Yaskawa INFORM job: DEMO_ROOF_UPPER_0625_3PAINT_69.JBI

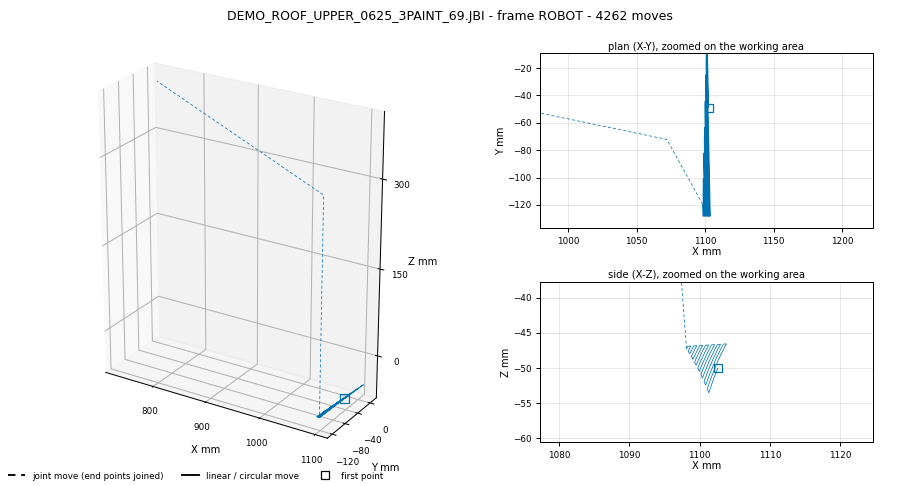
[picture p0: tool path of DEMO_ROOF_UPPER_0625_3PAINT_69.JBI in frame ROBOT, 4262 of 4262 moves have a stored position in this frame; points joined in program order, loops and branches not executed]
/JOB
//NAME DEMO_ROOF_UPPER_0625_3PAINT69
//POS
///NPOS 4262,0,0,0,0,0
///TOOL 0
///USER 0
///POSTYPE ROBOT
///RECTAN
///RCONF 1,0,0,0,0,0,0,0,0,0,0,0,0,0,0,0,0,0,0,0,0,0,0,0
C00000=1102.592,-48.864,-50.002,179.869,5.615,149.029
C00001=1102.586,-48.614,-50.014,179.869,5.619,149.030
C00002=1102.581,-48.364,-50.026,179.869,5.624,149.031
C00003=1102.575,-48.115,-50.039,179.869,5.629,149.032
C00004=1102.571,-47.865,-50.052,179.869,5.633,149.033
C00005=1102.566,-47.615,-50.065,179.868,5.638,149.034
C00006=1102.560,-47.366,-50.078,179.868,5.643,149.035
C00007=1102.555,-47.116,-50.090,179.868,5.648,149.037
C00008=1102.550,-46.866,-50.103,179.868,5.652,149.037
C00009=1102.545,-46.617,-50.115,179.868,5.657,149.039
C00010=1102.540,-46.368,-50.128,179.867,5.661,149.040
C00011=1102.534,-46.118,-50.141,179.868,5.666,149.041
C00012=1102.530,-45.904,-50.152,179.867,5.670,149.042
C00013=1102.526,-45.689,-50.162,179.867,5.674,149.043
C00014=1102.522,-45.475,-50.174,179.867,5.678,149.044
C00015=1102.517,-45.261,-50.184,179.867,5.683,149.045
C00016=1102.513,-45.047,-50.195,179.867,5.687,149.046
C00017=1102.508,-44.833,-50.206,179.867,5.691,149.046
C00018=1102.504,-44.618,-50.217,179.867,5.695,149.047
C00019=1102.500,-44.405,-50.228,179.866,5.699,149.048
C00020=1102.494,-44.154,-50.241,179.866,5.704,149.049
C00021=1102.489,-43.905,-50.253,179.866,5.708,149.050
C00022=1102.484,-43.656,-50.266,179.866,5.713,149.051
C00023=1102.479,-43.406,-50.279,179.866,5.718,149.053
C00024=1102.474,-43.157,-50.291,179.865,5.722,149.054
C00025=1102.468,-42.907,-50.305,179.866,5.727,149.055
C00026=1102.464,-42.657,-50.318,179.865,5.731,149.056
C00027=1102.459,-42.408,-50.330,179.865,5.737,149.057
C00028=1102.454,-42.158,-50.343,179.866,5.741,149.058
C00029=1102.449,-41.908,-50.356,179.866,5.746,149.059
C00030=1102.443,-41.659,-50.369,179.865,5.750,149.060
C00031=1102.438,-41.409,-50.382,179.865,5.756,149.061
C00032=1102.433,-41.160,-50.394,179.866,5.760,149.062
C00033=1102.428,-40.910,-50.407,179.866,5.765,149.063
C00034=1102.423,-40.660,-50.420,179.866,5.769,149.064
C00035=1102.417,-40.411,-50.433,179.865,5.774,149.065
C00036=1102.413,-40.161,-50.446,179.866,5.779,149.066
C00037=1102.407,-39.911,-50.459,179.866,5.783,149.067
C00038=1102.402,-39.662,-50.472,179.866,5.788,149.068
C00039=1102.397,-39.412,-50.485,179.866,5.793,149.069
C00040=1102.393,-39.163,-50.498,179.866,5.797,149.070
C00041=1102.387,-38.913,-50.512,179.866,5.802,149.071
C00042=1102.382,-38.664,-50.524,179.867,5.806,149.072
C00043=1102.377,-38.414,-50.537,179.867,5.811,149.073
C00044=1102.372,-38.164,-50.550,179.867,5.815,149.074
C00045=1102.367,-37.915,-50.563,179.867,5.820,149.075
C00046=1102.362,-37.665,-50.576,179.868,5.825,149.076
C00047=1102.356,-37.415,-50.589,179.867,5.829,149.077
C00048=1102.351,-37.166,-50.602,179.868,5.834,149.078
C00049=1102.346,-36.916,-50.616,179.868,5.837,149.079
C00050=1102.341,-36.667,-50.629,179.868,5.842,149.079
C00051=1102.336,-36.417,-50.641,179.869,5.847,149.080
C00052=1102.331,-36.167,-50.655,179.868,5.851,149.081
C00053=1102.326,-35.918,-50.667,179.869,5.856,149.082
C00054=1102.321,-35.668,-50.681,179.869,5.860,149.083
C00055=1102.316,-35.419,-50.694,179.869,5.864,149.084
C00056=1102.310,-35.169,-50.707,179.870,5.869,149.085
C00057=1102.305,-34.919,-50.720,179.870,5.874,149.086
C00058=1102.300,-34.670,-50.733,179.870,5.878,149.087
C00059=1102.296,-34.420,-50.747,179.870,5.882,149.088
C00060=1102.290,-34.171,-50.760,179.871,5.887,149.089
C00061=1102.285,-33.921,-50.773,179.871,5.891,149.089
C00062=1102.280,-33.671,-50.786,179.871,5.896,149.090
C00063=1102.275,-33.422,-50.799,179.872,5.901,149.091
C00064=1102.270,-33.172,-50.813,179.871,5.904,149.092
C00065=1102.264,-32.923,-50.825,179.872,5.909,149.093
C00066=1102.260,-32.673,-50.839,179.873,5.914,149.094
C00067=1102.254,-32.424,-50.852,179.873,5.917,149.095
C00068=1102.250,-32.209,-50.863,179.873,5.922,149.096
C00069=1102.246,-31.996,-50.875,179.874,5.926,149.096
C00070=1102.241,-31.781,-50.886,179.874,5.929,149.097
C00071=1102.237,-31.567,-50.898,179.874,5.933,149.098
C00072=1102.233,-31.353,-50.909,179.874,5.937,149.099
C00073=1102.229,-31.139,-50.921,179.875,5.941,149.099
C00074=1102.224,-30.925,-50.932,179.875,5.945,149.100
C00075=1102.220,-30.711,-50.944,179.875,5.949,149.101
C00076=1102.214,-30.461,-50.957,179.876,5.953,149.102
C00077=1102.210,-30.212,-50.971,179.876,5.957,149.103
C00078=1102.204,-29.962,-50.983,179.876,5.962,149.104
C00079=1102.199,-29.712,-50.997,179.876,5.967,149.104
C00080=1102.194,-29.463,-51.010,179.877,5.971,149.105
C00081=1102.189,-29.213,-51.024,179.877,5.975,149.106
C00082=1102.184,-28.964,-51.037,179.877,5.980,149.107
C00083=1102.179,-28.714,-51.051,179.878,5.984,149.108
C00084=1102.174,-28.465,-51.064,179.879,5.989,149.109
C00085=1102.169,-28.215,-51.078,179.879,5.994,149.110
C00086=1102.164,-27.966,-51.091,179.879,5.998,149.111
C00087=1102.159,-27.716,-51.105,179.879,6.003,149.112
C00088=1102.153,-27.467,-51.118,179.879,6.008,149.113
C00089=1102.149,-27.217,-51.131,179.880,6.012,149.114
C00090=1102.143,-26.967,-51.145,179.880,6.017,149.114
C00091=1102.139,-26.718,-51.158,179.881,6.022,149.115
C00092=1102.134,-26.468,-51.173,179.881,6.027,149.116
C00093=1102.128,-26.219,-51.186,179.881,6.030,149.117
C00094=1102.124,-25.969,-51.199,179.882,6.035,149.118
C00095=1102.118,-25.720,-51.213,179.882,6.040,149.119
C00096=1102.114,-25.470,-51.226,179.883,6.045,149.120
C00097=1102.108,-25.220,-51.240,179.883,6.050,149.121
C00098=1102.103,-24.971,-51.254,179.883,6.054,149.122
C00099=1102.098,-24.721,-51.267,179.883,6.058,149.123
C00100=1102.093,-24.472,-51.281,179.883,6.064,149.124
C00101=1102.088,-24.222,-51.295,179.883,6.068,149.125
C00102=1102.083,-23.972,-51.308,179.884,6.073,149.126
C00103=1102.078,-23.723,-51.322,179.884,6.078,149.127
C00104=1102.072,-23.473,-51.335,179.884,6.082,149.128
C00105=1102.068,-23.224,-51.349,179.884,6.087,149.129
C00106=1102.063,-22.974,-51.363,179.885,6.091,149.130
C00107=1102.057,-22.724,-51.377,179.885,6.096,149.131
C00108=1102.052,-22.475,-51.390,179.885,6.100,149.131
C00109=1102.048,-22.226,-51.404,179.886,6.105,149.132
C00110=1102.042,-21.975,-51.418,179.886,6.110,149.133
C00111=1102.037,-21.726,-51.432,179.886,6.115,149.134
C00112=1102.033,-21.477,-51.445,179.886,6.119,149.135
C00113=1102.027,-21.227,-51.458,179.886,6.123,149.136
C00114=1102.022,-20.977,-51.473,179.887,6.128,149.137
C00115=1102.017,-20.728,-51.487,179.887,6.133,149.138
C00116=1102.012,-20.478,-51.500,179.887,6.137,149.139
C00117=1102.007,-20.229,-51.514,179.888,6.141,149.140
C00118=1102.002,-19.979,-51.528,179.888,6.147,149.141
C00119=1101.996,-19.730,-51.542,179.888,6.151,149.142
C00120=1101.991,-19.480,-51.556,179.889,6.156,149.143
C00121=1101.987,-19.230,-51.569,179.889,6.160,149.144
C00122=1101.981,-18.981,-51.583,179.889,6.165,149.145
C00123=1101.976,-18.732,-51.598,179.890,6.169,149.145
C00124=1101.972,-18.518,-51.610,179.890,6.173,149.146
C00125=1101.967,-18.304,-51.622,179.890,6.177,149.147
C00126=1101.963,-18.090,-51.634,179.891,6.181,149.148
C00127=1101.959,-17.876,-51.645,179.891,6.185,149.149
C00128=1101.954,-17.662,-51.656,179.891,6.189,149.149
C00129=1101.950,-17.447,-51.669,179.891,6.192,149.150
C00130=1101.946,-17.233,-51.681,179.891,6.196,149.151
C00131=1101.942,-17.019,-51.693,179.892,6.200,149.152
C00132=1101.936,-16.770,-51.707,179.892,6.204,149.152
C00133=1101.931,-16.520,-51.721,179.893,6.209,149.153
C00134=1101.927,-16.271,-51.735,179.893,6.214,149.154
C00135=1101.922,-16.021,-51.749,179.894,6.218,149.155
C00136=1101.916,-15.772,-51.763,179.894,6.223,149.156
C00137=1101.911,-15.523,-51.777,179.894,6.227,149.157
C00138=1101.906,-15.273,-51.791,179.894,6.232,149.158
C00139=1101.901,-15.023,-51.805,179.895,6.237,149.159
C00140=1101.896,-14.774,-51.819,179.895,6.241,149.160
C00141=1101.891,-14.524,-51.833,179.896,6.246,149.161
C00142=1101.886,-14.274,-51.847,179.896,6.250,149.161
C00143=1101.881,-14.025,-51.861,179.897,6.254,149.162
C00144=1101.876,-13.776,-51.875,179.897,6.259,149.163
C00145=1101.871,-13.526,-51.889,179.898,6.264,149.164
C00146=1101.866,-13.276,-51.904,179.898,6.268,149.165
C00147=1101.861,-13.027,-51.918,179.898,6.272,149.166
C00148=1101.856,-12.777,-51.932,179.899,6.277,149.167
C00149=1101.850,-12.528,-51.946,179.899,6.282,149.168
C00150=1101.846,-12.278,-51.960,179.900,6.286,149.168
C00151=1101.841,-12.028,-51.975,179.900,6.290,149.169
C00152=1101.836,-11.779,-51.989,179.901,6.295,149.170
C00153=1101.831,-11.529,-52.003,179.901,6.299,149.171
C00154=1101.825,-11.280,-52.017,179.902,6.304,149.172
C00155=1101.820,-11.030,-52.031,179.902,6.309,149.173
C00156=1101.815,-10.781,-52.046,179.903,6.314,149.174
C00157=1101.811,-10.531,-52.061,179.903,6.317,149.174
C00158=1101.806,-10.282,-52.075,179.903,6.322,149.175
C00159=1101.801,-10.032,-52.089,179.904,6.327,149.176
C00160=1101.795,-9.783,-52.103,179.905,6.331,149.177
C00161=1101.790,-9.533,-52.117,179.905,6.336,149.178
C00162=1101.785,-9.284,-52.132,179.905,6.340,149.179
C00163=1101.780,-9.034,-52.146,179.906,6.344,149.179
C00164=1101.775,-8.784,-52.160,179.906,6.349,149.180
C00165=1101.770,-8.535,-52.175,179.907,6.354,149.181
C00166=1101.766,-8.285,-52.189,179.907,6.358,149.182
C00167=1101.760,-8.036,-52.203,179.908,6.363,149.183
C00168=1101.755,-7.787,-52.218,179.908,6.367,149.184
C00169=1101.750,-7.537,-52.232,179.909,6.371,149.185
C00170=1101.745,-7.287,-52.246,179.909,6.376,149.186
C00171=1101.741,-7.038,-52.261,179.910,6.380,149.186
C00172=1101.736,-6.788,-52.276,179.911,6.385,149.187
C00173=1101.730,-6.538,-52.290,179.911,6.390,149.188
C00174=1101.725,-6.289,-52.305,179.912,6.395,149.189
C00175=1101.720,-6.039,-52.319,179.912,6.398,149.190
C00176=1101.715,-5.791,-52.334,179.913,6.403,149.190
C00177=1101.710,-5.541,-52.348,179.913,6.408,149.191
C00178=1101.705,-5.291,-52.362,179.914,6.412,149.192
C00179=1101.700,-5.042,-52.377,179.915,6.417,149.193
C00180=1101.696,-4.828,-52.389,179.915,6.420,149.194
C00181=1101.691,-4.613,-52.402,179.916,6.425,149.194
C00182=1101.687,-4.400,-52.415,179.916,6.428,149.195
C00183=1101.683,-4.186,-52.427,179.916,6.432,149.196
C00184=1101.678,-3.973,-52.440,179.917,6.436,149.196
C00185=1101.675,-3.758,-52.452,179.918,6.440,149.197
C00186=1101.670,-3.544,-52.464,179.918,6.444,149.198
C00187=1101.666,-3.331,-52.477,179.919,6.448,149.199
C00188=1101.660,-3.081,-52.492,179.919,6.452,149.199
C00189=1101.656,-2.832,-52.507,179.920,6.456,149.200
C00190=1101.651,-2.582,-52.521,179.920,6.461,149.201
C00191=1101.646,-2.332,-52.535,179.921,6.466,149.202
C00192=1101.640,-2.083,-52.551,179.922,6.470,149.203
C00193=1101.635,-1.833,-52.565,179.922,6.475,149.204
C00194=1101.631,-1.584,-52.580,179.923,6.479,149.205
C00195=1101.626,-1.334,-52.594,179.924,6.484,149.205
C00196=1101.620,-1.084,-52.609,179.924,6.488,149.206
C00197=1101.615,-0.835,-52.624,179.925,6.493,149.207
C00198=1101.610,-0.586,-52.639,179.925,6.498,149.208
C00199=1101.606,-0.337,-52.654,179.926,6.502,149.209
C00200=1101.600,-0.086,-52.668,179.927,6.507,149.209
C00201=1101.595,0.163,-52.683,179.927,6.511,149.210
C00202=1101.590,0.412,-52.698,179.928,6.515,149.211
C00203=1101.586,0.661,-52.713,179.928,6.520,149.212
C00204=1101.580,0.911,-52.728,179.929,6.525,149.213
C00205=1101.575,1.161,-52.743,179.930,6.529,149.213
C00206=1101.571,1.410,-52.757,179.930,6.534,149.214
C00207=1101.565,1.660,-52.772,179.931,6.538,149.215
C00208=1101.560,1.909,-52.787,179.931,6.543,149.216
C00209=1101.556,2.158,-52.802,179.932,6.547,149.217
C00210=1101.550,2.408,-52.817,179.933,6.552,149.218
C00211=1101.545,2.658,-52.832,179.934,6.557,149.219
C00212=1101.541,2.907,-52.847,179.935,6.561,149.219
C00213=1101.535,3.157,-52.861,179.935,6.566,149.220
C00214=1101.530,3.406,-52.876,179.936,6.570,149.221
C00215=1101.526,3.656,-52.891,179.936,6.575,149.222
C00216=1101.520,3.906,-52.907,179.937,6.580,149.223
C00217=1101.516,4.155,-52.922,179.938,6.584,149.224
C00218=1101.510,4.405,-52.936,179.938,6.589,149.224
C00219=1101.505,4.654,-52.951,179.939,6.593,149.225
C00220=1101.501,4.903,-52.966,179.940,6.598,149.226
C00221=1101.495,5.153,-52.981,179.940,6.603,149.227
C00222=1101.490,5.402,-52.996,179.941,6.607,149.228
C00223=1101.485,5.651,-53.012,179.942,6.612,149.228
C00224=1101.480,5.901,-53.026,179.942,6.616,149.229
C00225=1101.475,6.151,-53.042,179.943,6.621,149.230
C00226=1101.471,6.400,-53.057,179.944,6.625,149.231
C00227=1101.466,6.649,-53.072,179.944,6.630,149.232
C00228=1101.460,6.899,-53.087,179.946,6.636,149.233
C00229=1101.456,7.148,-53.102,179.946,6.640,149.234
C00230=1101.450,7.398,-53.118,179.947,6.645,149.234
C00231=1101.446,7.647,-53.133,179.948,6.649,149.235
C00232=1101.441,7.898,-53.148,179.948,6.654,149.236
C00233=1101.436,8.147,-53.163,179.949,6.659,149.237
C00234=1101.431,8.396,-53.178,179.950,6.663,149.238
C00235=1101.426,8.645,-53.193,179.950,6.668,149.238
C00236=1101.419,8.979,-53.214,179.951,6.674,149.240
C00237=1101.412,9.313,-53.234,179.951,6.680,149.241
C00238=1101.406,9.648,-53.255,179.952,6.686,149.242
C00239=1101.399,9.982,-53.276,179.952,6.692,149.243
C00240=1101.394,10.231,-53.291,179.952,6.696,149.244
C00241=1101.388,10.481,-53.306,179.953,6.701,149.245
C00242=1101.384,10.730,-53.321,179.953,6.705,149.246
C00243=1101.379,10.980,-53.337,179.953,6.709,149.247
C00244=1101.374,11.229,-53.351,179.954,6.714,149.248
C00245=1101.369,11.478,-53.367,179.954,6.718,149.249
C00246=1101.364,11.728,-53.383,179.954,6.723,149.250
C00247=1101.359,11.978,-53.398,179.954,6.727,149.250
C00248=1101.354,12.227,-53.414,179.955,6.731,149.251
C00249=1101.349,12.476,-53.429,179.955,6.736,149.252
C00250=1101.344,12.725,-53.444,179.956,6.739,149.253
C00251=1101.339,12.975,-53.460,179.956,6.744,149.254
C00252=1101.335,13.225,-53.475,179.957,6.749,149.255
C00253=1101.329,13.474,-53.491,179.957,6.753,149.256
C00254=1101.325,13.723,-53.506,179.957,6.757,149.256
C00255=1101.319,13.973,-53.521,179.957,6.761,149.257
C00256=1101.094,4.203,-52.967,179.943,6.589,149.223
C00257=1101.098,3.953,-52.951,179.943,6.584,149.222
C00258=1101.102,3.704,-52.936,179.942,6.579,149.221
C00259=1101.108,3.454,-52.921,179.941,6.575,149.220
C00260=1101.113,3.205,-52.906,179.941,6.570,149.219
C00261=1101.118,2.956,-52.891,179.940,6.565,149.219
C00262=1101.123,2.706,-52.876,179.940,6.561,149.218
C00263=1101.128,2.457,-52.861,179.939,6.556,149.217
C00264=1101.133,2.207,-52.847,179.938,6.552,149.216
C00265=1101.138,1.958,-52.832,179.938,6.547,149.215
C00266=1101.143,1.709,-52.817,179.937,6.543,149.215
C00267=1101.148,1.459,-52.802,179.936,6.538,149.214
C00268=1101.153,1.209,-52.787,179.936,6.533,149.213
C00269=1101.158,0.960,-52.772,179.935,6.529,149.212
C00270=1101.163,0.710,-52.757,179.934,6.524,149.211
C00271=1101.168,0.461,-52.743,179.933,6.520,149.210
C00272=1101.173,0.212,-52.728,179.933,6.515,149.209
C00273=1101.178,-0.039,-52.712,179.932,6.511,149.209
C00274=1101.183,-0.288,-52.697,179.931,6.506,149.208
C00275=1101.188,-0.538,-52.683,179.931,6.501,149.207
C00276=1101.192,-0.787,-52.668,179.930,6.497,149.206
C00277=1101.198,-1.037,-52.653,179.929,6.492,149.205
C00278=1101.203,-1.286,-52.638,179.929,6.487,149.205
C00279=1101.208,-1.536,-52.624,179.928,6.483,149.204
C00280=1101.212,-1.785,-52.609,179.927,6.478,149.203
C00281=1101.218,-2.035,-52.594,179.927,6.474,149.202
C00282=1101.223,-2.285,-52.580,179.927,6.470,149.201
C00283=1101.228,-2.534,-52.565,179.926,6.465,149.201
C00284=1101.233,-2.783,-52.551,179.925,6.461,149.200
C00285=1101.239,-3.032,-52.535,179.925,6.456,149.199
C00286=1101.244,-3.282,-52.521,179.924,6.452,149.198
C00287=1101.248,-3.532,-52.507,179.923,6.447,149.197
C00288=1101.253,-3.781,-52.492,179.923,6.442,149.196
C00289=1101.260,-4.095,-52.474,179.922,6.436,149.195
C00290=1101.266,-4.408,-52.455,179.921,6.431,149.194
C00291=1101.273,-4.721,-52.437,179.921,6.426,149.193
C00292=1101.278,-5.034,-52.419,179.920,6.420,149.192
C00293=1101.283,-5.284,-52.404,179.919,6.415,149.191
C00294=1101.288,-5.533,-52.389,179.919,6.411,149.190
C00295=1101.294,-5.783,-52.374,179.918,6.406,149.190
C00296=1101.299,-6.033,-52.360,179.918,6.401,149.189
C00297=1101.304,-6.283,-52.346,179.917,6.397,149.188
C00298=1101.308,-6.532,-52.331,179.916,6.392,149.187
C00299=1101.314,-6.781,-52.317,179.916,6.388,149.186
C00300=1101.319,-7.030,-52.303,179.916,6.384,149.185
C00301=1101.324,-7.280,-52.288,179.915,6.379,149.185
C00302=1101.328,-7.529,-52.273,179.914,6.375,149.184
C00303=1101.333,-7.779,-52.259,179.914,6.370,149.183
C00304=1101.339,-8.029,-52.244,179.913,6.365,149.182
C00305=1101.344,-8.279,-52.230,179.913,6.362,149.181
C00306=1101.349,-8.528,-52.216,179.912,6.357,149.180
C00307=1101.354,-8.777,-52.201,179.912,6.352,149.179
C00308=1101.359,-9.026,-52.187,179.911,6.348,149.179
C00309=1101.364,-9.276,-52.173,179.911,6.343,149.178
C00310=1101.369,-9.526,-52.158,179.910,6.338,149.177
C00311=1101.374,-9.776,-52.144,179.910,6.335,149.176
C00312=1101.379,-10.025,-52.130,179.910,6.330,149.175
C00313=1101.384,-10.275,-52.115,179.909,6.325,149.174
C00314=1101.389,-10.524,-52.100,179.909,6.320,149.173
C00315=1101.394,-10.773,-52.087,179.908,6.316,149.173
C00316=1101.399,-11.023,-52.072,179.908,6.312,149.172
C00317=1101.404,-11.273,-52.058,179.907,6.307,149.171
C00318=1101.409,-11.522,-52.044,179.907,6.303,149.170
C00319=1101.414,-11.772,-52.029,179.906,6.298,149.169
C00320=1101.419,-12.022,-52.015,179.906,6.293,149.168
C00321=1101.424,-12.271,-52.001,179.905,6.290,149.168
C00322=1101.429,-12.520,-51.987,179.905,6.285,149.167
C00323=1101.434,-12.770,-51.973,179.904,6.280,149.166
C00324=1101.439,-13.020,-51.958,179.904,6.276,149.165
C00325=1101.444,-13.270,-51.944,179.903,6.271,149.164
C00326=1101.450,-13.519,-51.930,179.903,6.267,149.163
C00327=1101.455,-13.768,-51.916,179.903,6.262,149.162
C00328=1101.460,-14.018,-51.902,179.902,6.258,149.161
C00329=1101.464,-14.267,-51.888,179.901,6.253,149.161
C00330=1101.469,-14.517,-51.874,179.901,6.248,149.160
C00331=1101.474,-14.766,-51.860,179.901,6.245,149.159
C00332=1101.479,-15.016,-51.846,179.901,6.240,149.158
C00333=1101.484,-15.265,-51.831,179.900,6.235,149.157
C00334=1101.489,-15.515,-51.817,179.900,6.230,149.156
C00335=1101.495,-15.764,-51.803,179.899,6.226,149.155
C00336=1101.500,-16.014,-51.789,179.899,6.222,149.154
C00337=1101.505,-16.264,-51.775,179.899,6.217,149.153
C00338=1101.509,-16.514,-51.762,179.898,6.212,149.152
C00339=1101.515,-16.763,-51.748,179.898,6.208,149.152
C00340=1101.520,-17.012,-51.733,179.898,6.204,149.151
C00341=1101.524,-17.226,-51.721,179.897,6.199,149.150
C00342=1101.529,-17.440,-51.709,179.897,6.195,149.149
C00343=1101.533,-17.654,-51.697,179.897,6.192,149.148
C00344=1101.538,-17.868,-51.685,179.896,6.188,149.148
C00345=1101.542,-18.082,-51.673,179.896,6.184,149.147
C00346=1101.546,-18.296,-51.662,179.895,6.180,149.146
C00347=1101.550,-18.510,-51.649,179.895,6.176,149.145
C00348=1101.554,-18.724,-51.637,179.895,6.173,149.145
C00349=1101.560,-18.973,-51.623,179.895,6.168,149.144
C00350=1101.565,-19.223,-51.609,179.894,6.163,149.143
C00351=1101.570,-19.473,-51.596,179.894,6.159,149.142
C00352=1101.575,-19.722,-51.582,179.894,6.154,149.141
C00353=1101.580,-19.972,-51.568,179.894,6.149,149.140
C00354=1101.585,-20.221,-51.554,179.893,6.145,149.139
C00355=1101.590,-20.470,-51.540,179.893,6.140,149.138
C00356=1101.595,-20.721,-51.526,179.893,6.136,149.137
C00357=1101.600,-20.970,-51.513,179.892,6.131,149.136
C00358=1101.605,-21.219,-51.499,179.892,6.127,149.135
C00359=1101.610,-21.469,-51.485,179.891,6.122,149.134
C00360=1101.615,-21.719,-51.471,179.892,6.118,149.133
C00361=1101.620,-21.968,-51.458,179.892,6.113,149.132
C00362=1101.625,-22.218,-51.443,179.891,6.108,149.131
C00363=1101.630,-22.468,-51.430,179.891,6.103,149.131
C00364=1101.635,-22.717,-51.416,179.891,6.099,149.130
C00365=1101.640,-22.966,-51.402,179.890,6.095,149.129
C00366=1101.646,-23.216,-51.389,179.890,6.090,149.128
C00367=1101.651,-23.466,-51.375,179.890,6.085,149.127
C00368=1101.655,-23.715,-51.361,179.890,6.081,149.126
C00369=1101.661,-23.965,-51.348,179.889,6.076,149.125
C00370=1101.666,-24.214,-51.333,179.889,6.072,149.124
C00371=1101.671,-24.464,-51.320,179.889,6.066,149.123
C00372=1101.676,-24.713,-51.307,179.889,6.062,149.122
C00373=1101.681,-24.963,-51.292,179.889,6.058,149.121
C00374=1101.686,-25.212,-51.280,179.888,6.053,149.120
C00375=1101.691,-25.462,-51.265,179.888,6.048,149.119
C00376=1101.696,-25.712,-51.252,179.888,6.044,149.118
C00377=1101.701,-25.961,-51.239,179.888,6.039,149.117
C00378=1101.707,-26.211,-51.225,179.887,6.035,149.116
C00379=1101.712,-26.460,-51.211,179.887,6.030,149.115
C00380=1101.716,-26.710,-51.197,179.886,6.025,149.114
C00381=1101.722,-26.960,-51.184,179.886,6.020,149.113
C00382=1101.726,-27.209,-51.170,179.886,6.015,149.112
C00383=1101.732,-27.459,-51.157,179.885,6.011,149.111
C00384=1101.737,-27.708,-51.143,179.885,6.006,149.111
C00385=1101.742,-27.958,-51.130,179.885,6.001,149.110
C00386=1101.747,-28.207,-51.116,179.885,5.997,149.109
C00387=1101.752,-28.457,-51.103,179.884,5.992,149.108
C00388=1101.757,-28.706,-51.089,179.884,5.988,149.107
C00389=1101.762,-28.956,-51.076,179.883,5.983,149.106
C00390=1101.768,-29.206,-51.063,179.882,5.979,149.105
C00391=1101.773,-29.456,-51.049,179.882,5.975,149.104
C00392=1101.778,-29.705,-51.036,179.882,5.970,149.104
C00393=1101.783,-29.955,-51.022,179.882,5.965,149.103
C00394=1101.787,-30.205,-51.009,179.881,5.960,149.102
C00395=1101.793,-30.454,-50.995,179.881,5.956,149.101
C00396=1101.797,-30.704,-50.982,179.881,5.952,149.100
C00397=1101.802,-30.917,-50.970,179.880,5.948,149.099
C00398=1101.806,-31.131,-50.960,179.880,5.944,149.098
C00399=1101.811,-31.345,-50.948,179.880,5.940,149.098
C00400=1101.816,-31.560,-50.936,179.879,5.936,149.097
C00401=1101.819,-31.773,-50.925,179.879,5.933,149.096
C00402=1101.824,-31.988,-50.914,179.879,5.929,149.095
C00403=1101.828,-32.201,-50.902,179.878,5.925,149.095
C00404=1101.833,-32.416,-50.891,179.878,5.921,149.094
C00405=1101.838,-32.665,-50.878,179.878,5.917,149.093
C00406=1101.843,-32.915,-50.864,179.878,5.912,149.092
C00407=1101.848,-33.164,-50.851,179.877,5.908,149.091
C00408=1101.853,-33.414,-50.837,179.877,5.904,149.090
C00409=1101.858,-33.663,-50.825,179.877,5.899,149.089
C00410=1101.863,-33.914,-50.811,179.876,5.894,149.089
C00411=1101.868,-34.163,-50.798,179.876,5.890,149.088
C00412=1101.873,-34.413,-50.784,179.876,5.886,149.087
C00413=1101.878,-34.662,-50.771,179.875,5.881,149.086
C00414=1101.884,-34.911,-50.759,179.876,5.877,149.085
C00415=1101.889,-35.162,-50.745,179.875,5.872,149.084
C00416=1101.894,-35.410,-50.732,179.875,5.868,149.083
C00417=1101.899,-35.661,-50.718,179.875,5.864,149.082
C00418=1101.904,-35.910,-50.706,179.874,5.859,149.081
C00419=1101.909,-36.160,-50.693,179.874,5.854,149.080
C00420=1101.914,-36.409,-50.679,179.874,5.850,149.079
C00421=1101.919,-36.658,-50.666,179.874,5.845,149.078
C00422=1101.924,-36.909,-50.653,179.873,5.841,149.078
C00423=1101.930,-37.158,-50.640,179.873,5.837,149.077
C00424=1101.934,-37.408,-50.627,179.873,5.832,149.076
C00425=1101.940,-37.658,-50.614,179.873,5.828,149.075
C00426=1101.945,-37.906,-50.601,179.873,5.823,149.074
C00427=1101.949,-38.156,-50.588,179.872,5.819,149.073
C00428=1101.955,-38.406,-50.575,179.873,5.814,149.072
C00429=1101.960,-38.656,-50.562,179.872,5.810,149.071
C00430=1101.965,-38.905,-50.549,179.872,5.805,149.070
C00431=1101.971,-39.155,-50.536,179.872,5.801,149.069
C00432=1101.975,-39.405,-50.523,179.872,5.796,149.068
C00433=1101.980,-39.654,-50.510,179.872,5.791,149.067
C00434=1101.986,-39.903,-50.496,179.872,5.787,149.066
C00435=1101.990,-40.153,-50.483,179.871,5.782,149.065
C00436=1101.996,-40.403,-50.471,179.871,5.777,149.064
C00437=1102.001,-40.652,-50.458,179.872,5.773,149.063
C00438=1102.006,-40.902,-50.445,179.872,5.768,149.062
C00439=1102.011,-41.152,-50.432,179.871,5.764,149.061
C00440=1102.016,-41.401,-50.419,179.872,5.759,149.060
C00441=1102.021,-41.651,-50.406,179.871,5.754,149.059
C00442=1102.027,-41.901,-50.393,179.872,5.749,149.058
C00443=1102.032,-42.150,-50.381,179.871,5.745,149.057
C00444=1102.036,-42.400,-50.368,179.872,5.740,149.056
C00445=1102.042,-42.650,-50.354,179.871,5.736,149.055
C00446=1102.047,-42.899,-50.342,179.871,5.730,149.054
C00447=1102.052,-43.149,-50.329,179.872,5.726,149.053
C00448=1102.057,-43.398,-50.316,179.872,5.721,149.051
C00449=1102.063,-43.648,-50.303,179.872,5.716,149.051
C00450=1102.067,-43.898,-50.290,179.872,5.712,149.049
C00451=1102.072,-44.147,-50.278,179.872,5.707,149.048
C00452=1102.077,-44.396,-50.265,179.873,5.703,149.047
C00453=1102.082,-44.611,-50.254,179.873,5.698,149.046
C00454=1102.086,-44.825,-50.243,179.873,5.694,149.045
C00455=1102.090,-45.040,-50.232,179.873,5.690,149.044
C00456=1102.096,-45.253,-50.221,179.873,5.686,149.043
C00457=1102.100,-45.468,-50.210,179.873,5.682,149.043
C00458=1102.103,-45.681,-50.199,179.873,5.678,149.042
C00459=1102.108,-45.896,-50.188,179.874,5.674,149.041
C00460=1102.113,-46.109,-50.177,179.874,5.670,149.040
C00461=1102.117,-46.359,-50.164,179.874,5.665,149.039
C00462=1102.122,-46.609,-50.152,179.873,5.660,149.038
C00463=1102.128,-46.859,-50.140,179.874,5.656,149.037
C00464=1102.134,-47.108,-50.127,179.874,5.651,149.035
C00465=1102.138,-47.358,-50.114,179.874,5.646,149.034
C00466=1102.143,-47.608,-50.101,179.874,5.642,149.033
C00467=1102.149,-47.857,-50.089,179.874,5.637,149.032
C00468=1102.154,-48.106,-50.076,179.875,5.632,149.031
C00469=1102.159,-48.357,-50.064,179.875,5.628,149.030
C00470=1102.164,-48.606,-50.051,179.875,5.623,149.029
C00471=1102.169,-48.855,-50.039,179.875,5.618,149.028
C00472=1102.175,-49.105,-50.025,179.876,5.613,149.027
C00473=1102.179,-49.355,-50.012,179.875,5.608,149.026
C00474=1102.185,-49.605,-50.000,179.876,5.604,149.025
C00475=1102.190,-49.854,-49.988,179.876,5.599,149.023
C00476=1102.195,-50.104,-49.975,179.875,5.594,149.022
C00477=1102.200,-50.353,-49.963,179.876,5.590,149.021
C00478=1102.204,-50.603,-49.950,179.876,5.585,149.020
C00479=1102.210,-50.853,-49.938,179.876,5.580,149.019
C00480=1102.215,-51.102,-49.925,179.876,5.576,149.018
C00481=1102.220,-51.352,-49.913,179.877,5.571,149.017
C00482=1102.226,-51.602,-49.901,179.876,5.566,149.016
C00483=1102.230,-51.852,-49.888,179.877,5.562,149.015
C00484=1102.235,-52.101,-49.875,179.877,5.556,149.014
C00485=1102.240,-52.350,-49.863,179.876,5.552,149.013
C00486=1102.246,-52.600,-49.851,179.877,5.547,149.012
C00487=1102.251,-52.849,-49.838,179.877,5.542,149.010
C00488=1102.256,-53.099,-49.825,179.877,5.538,149.010
C00489=1102.261,-53.349,-49.813,179.877,5.533,149.008
C00490=1102.266,-53.599,-49.801,179.878,5.528,149.007
C00491=1102.271,-53.848,-49.788,179.877,5.523,149.006
C00492=1102.277,-54.098,-49.776,179.878,5.519,149.005
C00493=1102.282,-54.347,-49.764,179.877,5.514,149.004
C00494=1102.287,-54.597,-49.751,179.878,5.509,149.003
C00495=1102.292,-54.847,-49.739,179.878,5.505,149.002
C00496=1102.297,-55.097,-49.726,179.878,5.500,149.001
C00497=1102.302,-55.346,-49.714,179.878,5.495,149.000
C00498=1102.307,-55.596,-49.702,179.879,5.491,148.999
C00499=1102.312,-55.845,-49.689,179.878,5.486,148.998
C00500=1102.318,-56.095,-49.677,179.878,5.481,148.997
C00501=1102.323,-56.344,-49.665,179.878,5.477,148.996
C00502=1102.328,-56.594,-49.653,179.879,5.472,148.995
C00503=1102.333,-56.844,-49.640,179.879,5.467,148.993
C00504=1102.338,-57.094,-49.628,179.879,5.463,148.992
C00505=1102.343,-57.344,-49.615,179.879,5.458,148.991
C00506=1102.349,-57.593,-49.603,179.879,5.453,148.990
C00507=1102.353,-57.843,-49.591,179.879,5.448,148.989
C00508=1102.358,-58.092,-49.579,179.879,5.443,148.988
C00509=1102.363,-58.307,-49.569,179.879,5.440,148.987
C00510=1102.368,-58.521,-49.558,179.879,5.435,148.986
C00511=1102.372,-58.735,-49.547,179.879,5.431,148.985
C00512=1102.376,-58.949,-49.536,179.879,5.427,148.985
C00513=1102.381,-59.163,-49.527,179.879,5.423,148.984
C00514=1102.385,-59.377,-49.516,179.879,5.419,148.983
C00515=1102.389,-59.592,-49.505,179.880,5.415,148.982
C00516=1102.394,-59.806,-49.496,179.879,5.411,148.981
C00517=1102.399,-60.055,-49.483,179.879,5.407,148.980
C00518=1102.405,-60.305,-49.471,179.880,5.401,148.979
C00519=1102.410,-60.554,-49.458,179.879,5.397,148.978
C00520=1102.415,-60.805,-49.446,179.879,5.392,148.977
C00521=1102.419,-61.054,-49.434,179.879,5.387,148.976
C00522=1102.424,-61.304,-49.422,179.879,5.382,148.975
C00523=1102.430,-61.553,-49.410,179.879,5.377,148.974
C00524=1102.435,-61.803,-49.398,179.879,5.372,148.972
C00525=1102.440,-62.053,-49.386,179.878,5.367,148.972
C00526=1102.445,-62.302,-49.374,179.878,5.362,148.970
C00527=1102.450,-62.552,-49.362,179.878,5.357,148.969
C00528=1102.456,-62.802,-49.350,179.878,5.352,148.968
C00529=1102.461,-63.051,-49.338,179.878,5.347,148.967
C00530=1102.465,-63.301,-49.326,179.878,5.342,148.966
C00531=1102.471,-63.551,-49.314,179.877,5.337,148.965
C00532=1102.476,-63.800,-49.302,179.878,5.332,148.964
C00533=1102.481,-64.050,-49.290,179.878,5.328,148.963
C00534=1102.487,-64.300,-49.278,179.878,5.323,148.962
C00535=1102.491,-64.549,-49.266,179.878,5.318,148.961
C00536=1102.497,-64.799,-49.254,179.878,5.313,148.960
C00537=1102.502,-65.049,-49.242,179.878,5.308,148.959
C00538=1102.507,-65.298,-49.230,179.878,5.303,148.958
C00539=1102.512,-65.548,-49.218,179.878,5.298,148.956
C00540=1102.517,-65.798,-49.206,179.878,5.293,148.955
C00541=1102.523,-66.048,-49.195,179.878,5.288,148.954
C00542=1102.527,-66.297,-49.183,179.878,5.283,148.953
C00543=1102.533,-66.547,-49.171,179.878,5.278,148.952
C00544=1102.538,-66.797,-49.159,179.878,5.273,148.951
C00545=1102.543,-67.046,-49.148,179.878,5.268,148.950
C00546=1102.548,-67.295,-49.135,179.878,5.263,148.949
C00547=1102.554,-67.545,-49.123,179.878,5.258,148.948
C00548=1102.559,-67.794,-49.112,179.878,5.253,148.947
C00549=1102.564,-68.044,-49.100,179.878,5.248,148.945
C00550=1102.569,-68.294,-49.088,179.878,5.243,148.944
C00551=1102.574,-68.544,-49.077,179.878,5.238,148.943
C00552=1102.579,-68.793,-49.064,179.878,5.233,148.942
C00553=1102.585,-69.043,-49.053,179.878,5.228,148.941
C00554=1102.589,-69.293,-49.041,179.878,5.223,148.940
C00555=1102.595,-69.543,-49.029,179.878,5.217,148.939
C00556=1102.599,-69.792,-49.018,179.878,5.212,148.937
C00557=1102.605,-70.042,-49.006,179.878,5.207,148.936
C00558=1102.611,-70.292,-48.995,179.878,5.202,148.935
C00559=1102.616,-70.541,-48.983,179.878,5.197,148.934
C00560=1102.621,-70.791,-48.971,179.878,5.192,148.933
C00561=1102.626,-71.040,-48.959,179.878,5.187,148.932
C00562=1102.631,-71.290,-48.948,179.878,5.182,148.931
C00563=1102.636,-71.540,-48.936,179.879,5.177,148.930
C00564=1102.641,-71.790,-48.924,179.879,5.172,148.928
C00565=1102.646,-72.004,-48.915,179.879,5.168,148.927
C00566=1102.650,-72.219,-48.905,179.879,5.164,148.926
C00567=1102.655,-72.432,-48.894,179.879,5.159,148.925
C00568=1102.659,-72.647,-48.884,179.880,5.155,148.924
C00569=1102.664,-72.861,-48.875,179.879,5.150,148.923
C00570=1102.667,-73.075,-48.865,179.879,5.146,148.923
C00571=1102.672,-73.289,-48.855,179.880,5.142,148.921
C00572=1102.677,-73.504,-48.845,179.880,5.137,148.920
C00573=1102.683,-73.753,-48.834,179.880,5.132,148.919
C00574=1102.687,-74.003,-48.822,179.880,5.127,148.918
C00575=1102.693,-74.253,-48.810,179.880,5.121,148.917
C00576=1102.698,-74.503,-48.799,179.880,5.116,148.916
C00577=1102.703,-74.753,-48.787,179.881,5.111,148.915
C00578=1102.708,-75.001,-48.776,179.881,5.106,148.913
C00579=1102.714,-75.251,-48.764,179.881,5.101,148.912
C00580=1102.718,-75.501,-48.753,179.881,5.096,148.911
C00581=1102.724,-75.751,-48.741,179.882,5.091,148.910
C00582=1102.729,-76.001,-48.730,179.882,5.086,148.909
C00583=1102.735,-76.250,-48.718,179.882,5.081,148.907
C00584=1102.739,-76.499,-48.707,179.882,5.076,148.906
C00585=1102.745,-76.750,-48.696,179.882,5.071,148.905
C00586=1102.750,-77.000,-48.685,179.882,5.066,148.904
C00587=1102.754,-77.249,-48.673,179.883,5.061,148.903
C00588=1102.760,-77.498,-48.662,179.883,5.056,148.902
C00589=1102.765,-77.748,-48.651,179.883,5.050,148.900
C00590=1102.771,-77.998,-48.639,179.883,5.045,148.899
C00591=1102.775,-78.248,-48.627,179.883,5.040,148.898
C00592=1102.782,-78.497,-48.617,179.884,5.035,148.897
C00593=1102.786,-78.747,-48.605,179.884,5.029,148.895
C00594=1102.791,-78.997,-48.594,179.884,5.024,148.894
C00595=1102.796,-79.247,-48.582,179.884,5.019,148.893
C00596=1102.802,-79.496,-48.571,179.885,5.014,148.892
C00597=1102.807,-79.746,-48.560,179.885,5.009,148.891
C00598=1102.812,-79.996,-48.549,179.885,5.004,148.890
C00599=1102.817,-80.245,-48.537,179.885,4.999,148.888
C00600=1102.823,-80.495,-48.526,179.886,4.994,148.887
C00601=1102.828,-80.744,-48.515,179.886,4.989,148.886
C00602=1102.833,-80.995,-48.503,179.886,4.984,148.885
C00603=1102.839,-81.244,-48.493,179.886,4.979,148.884
C00604=1102.843,-81.493,-48.481,179.887,4.973,148.882
C00605=1102.849,-81.744,-48.470,179.887,4.968,148.881
C00606=1102.854,-81.994,-48.459,179.887,4.963,148.880
C00607=1102.859,-82.242,-48.448,179.887,4.958,148.879
C00608=1102.864,-82.492,-48.436,179.888,4.953,148.878
C00609=1102.869,-82.743,-48.425,179.888,4.948,148.876
C00610=1102.875,-82.992,-48.414,179.888,4.943,148.875
C00611=1102.879,-83.241,-48.403,179.889,4.938,148.874
C00612=1102.885,-83.492,-48.392,179.889,4.933,148.873
C00613=1102.890,-83.741,-48.381,179.889,4.928,148.872
C00614=1102.895,-83.990,-48.370,179.890,4.922,148.870
C00615=1102.901,-84.241,-48.359,179.890,4.917,148.869
C00616=1102.906,-84.490,-48.348,179.890,4.912,148.868
C00617=1102.911,-84.739,-48.336,179.890,4.907,148.867
C00618=1102.916,-84.990,-48.326,179.890,4.902,148.865
C00619=1102.922,-85.239,-48.314,179.891,4.897,148.864
C00620=1102.927,-85.489,-48.304,179.891,4.892,148.863
C00621=1102.932,-85.703,-48.294,179.892,4.887,148.862
C00622=1102.935,-85.918,-48.285,179.892,4.883,148.861
C00623=1102.940,-86.132,-48.275,179.892,4.879,148.860
C00624=1102.944,-86.347,-48.266,179.892,4.874,148.859
C00625=1102.949,-86.561,-48.256,179.892,4.870,148.858
C00626=1102.953,-86.775,-48.247,179.893,4.866,148.857
C00627=1102.957,-86.989,-48.237,179.893,4.861,148.856
C00628=1102.962,-87.204,-48.227,179.893,4.857,148.855
C00629=1102.967,-87.454,-48.217,179.893,4.852,148.854
C00630=1102.973,-87.703,-48.206,179.894,4.847,148.852
C00631=1102.978,-87.953,-48.195,179.894,4.843,148.851
C00632=1102.983,-88.202,-48.184,179.895,4.837,148.850
C00633=1102.989,-88.452,-48.173,179.895,4.832,148.849
C00634=1102.993,-88.702,-48.162,179.895,4.827,148.847
C00635=1102.999,-88.952,-48.152,179.896,4.822,148.846
C00636=1103.004,-89.201,-48.140,179.896,4.817,148.845
C00637=1103.009,-89.451,-48.130,179.897,4.812,148.844
C00638=1103.014,-89.700,-48.119,179.897,4.807,148.843
C00639=1103.020,-89.951,-48.108,179.897,4.802,148.842
C00640=1103.025,-90.200,-48.097,179.897,4.797,148.840
C00641=1103.030,-90.450,-48.086,179.898,4.792,148.839
C00642=1103.035,-90.699,-48.075,179.898,4.787,148.838
C00643=1103.040,-90.949,-48.065,179.898,4.782,148.837
C00644=1103.045,-91.200,-48.054,179.898,4.777,148.836
C00645=1103.051,-91.448,-48.043,179.899,4.772,148.834
C00646=1103.056,-91.699,-48.033,179.899,4.767,148.833
C00647=1103.062,-91.948,-48.021,179.900,4.762,148.832
C00648=1103.067,-92.198,-48.011,179.900,4.757,148.831
C00649=1103.072,-92.447,-48.000,179.901,4.752,148.829
C00650=1103.077,-92.697,-47.989,179.901,4.747,148.828
C00651=1103.082,-92.947,-47.979,179.902,4.742,148.827
C00652=1103.087,-93.197,-47.968,179.902,4.737,148.826
C00653=1103.092,-93.447,-47.957,179.903,4.733,148.825
C00654=1103.098,-93.696,-47.947,179.903,4.728,148.823
C00655=1103.102,-93.946,-47.935,179.903,4.722,148.822
C00656=1103.108,-94.196,-47.925,179.903,4.717,148.821
C00657=1103.113,-94.446,-47.915,179.904,4.713,148.820
C00658=1103.118,-94.695,-47.904,179.904,4.708,148.819
C00659=1103.123,-94.945,-47.893,179.904,4.703,148.817
C00660=1103.129,-95.194,-47.883,179.905,4.698,148.816
C00661=1103.134,-95.444,-47.871,179.905,4.693,148.815
C00662=1103.140,-95.694,-47.861,179.906,4.688,148.814
C00663=1103.145,-95.944,-47.850,179.906,4.684,148.813
C00664=1103.150,-96.193,-47.839,179.907,4.679,148.811
C00665=1103.155,-96.443,-47.829,179.907,4.673,148.810
C00666=1103.161,-96.693,-47.819,179.908,4.669,148.809
C00667=1103.166,-96.943,-47.808,179.908,4.664,148.808
C00668=1103.171,-97.192,-47.797,179.908,4.659,148.807
C00669=1103.176,-97.442,-47.787,179.909,4.654,148.806
C00670=1103.182,-97.692,-47.776,179.909,4.649,148.804
C00671=1103.187,-97.942,-47.766,179.909,4.644,148.803
C00672=1103.192,-98.191,-47.755,179.910,4.640,148.802
C00673=1103.198,-98.441,-47.745,179.910,4.635,148.801
C00674=1103.203,-98.691,-47.734,179.910,4.630,148.800
C00675=1103.208,-98.940,-47.724,179.911,4.624,148.798
C00676=1103.212,-99.190,-47.714,179.911,4.620,148.797
C00677=1103.217,-99.404,-47.704,179.912,4.616,148.796
C00678=1103.222,-99.619,-47.696,179.912,4.611,148.795
C00679=1103.226,-99.834,-47.686,179.912,4.607,148.794
C00680=1103.231,-100.048,-47.678,179.913,4.603,148.793
C00681=1103.235,-100.262,-47.669,179.913,4.599,148.792
C00682=1103.240,-100.477,-47.660,179.914,4.595,148.791
C00683=1103.244,-100.691,-47.651,179.914,4.591,148.790
C00684=1103.248,-100.906,-47.642,179.914,4.586,148.789
C00685=1103.254,-101.155,-47.631,179.915,4.581,148.788
C00686=1103.259,-101.404,-47.621,179.915,4.576,148.786
C00687=1103.264,-101.655,-47.610,179.915,4.571,148.785
C00688=1103.270,-101.904,-47.600,179.916,4.567,148.784
C00689=1103.275,-102.154,-47.589,179.916,4.562,148.783
C00690=1103.280,-102.404,-47.579,179.917,4.556,148.782
C00691=1103.286,-102.653,-47.569,179.917,4.551,148.780
C00692=1103.291,-102.904,-47.558,179.918,4.547,148.779
C00693=1103.296,-103.153,-47.549,179.918,4.542,148.778
C00694=1103.301,-103.403,-47.538,179.918,4.537,148.777
C00695=1103.306,-103.652,-47.527,179.919,4.532,148.776
C00696=1103.312,-103.902,-47.517,179.919,4.527,148.774
C00697=1103.317,-104.152,-47.506,179.919,4.522,148.773
C00698=1103.322,-104.401,-47.496,179.920,4.516,148.772
C00699=1103.327,-104.652,-47.486,179.921,4.512,148.770
C00700=1103.332,-104.901,-47.476,179.921,4.507,148.769
C00701=1103.338,-105.150,-47.466,179.921,4.502,148.768
C00702=1103.343,-105.401,-47.455,179.922,4.497,148.767
C00703=1103.348,-105.650,-47.445,179.923,4.492,148.766
C00704=1103.353,-105.901,-47.434,179.923,4.487,148.764
C00705=1103.358,-106.150,-47.425,179.923,4.482,148.763
C00706=1103.364,-106.399,-47.415,179.924,4.478,148.762
C00707=1103.369,-106.650,-47.404,179.924,4.473,148.761
C00708=1103.374,-106.899,-47.394,179.925,4.467,148.759
C00709=1103.380,-107.149,-47.384,179.925,4.462,148.758
C00710=1103.384,-107.399,-47.374,179.926,4.458,148.757
C00711=1103.390,-107.648,-47.363,179.926,4.452,148.756
C00712=1103.395,-107.898,-47.353,179.926,4.447,148.755
C00713=1103.400,-108.148,-47.343,179.927,4.442,148.753
C00714=1103.406,-108.397,-47.333,179.927,4.438,148.752
C00715=1103.411,-108.647,-47.324,179.928,4.433,148.751
C00716=1103.416,-108.898,-47.313,179.928,4.427,148.750
C00717=1103.422,-109.147,-47.303,179.929,4.422,148.748
C00718=1103.427,-109.396,-47.293,179.929,4.418,148.747
C00719=1103.432,-109.647,-47.283,179.930,4.412,148.746
C00720=1103.437,-109.896,-47.272,179.930,4.407,148.745
C00721=1103.443,-110.146,-47.262,179.930,4.402,148.743
C00722=1103.448,-110.395,-47.253,179.932,4.397,148.742
C00723=1103.453,-110.645,-47.242,179.932,4.392,148.741
C00724=1103.459,-110.895,-47.233,179.932,4.387,148.740
C00725=1103.464,-111.145,-47.222,179.932,4.382,148.738
C00726=1103.469,-111.395,-47.212,179.933,4.377,148.737
C00727=1103.474,-111.644,-47.202,179.933,4.372,148.736
C00728=1103.480,-111.894,-47.192,179.934,4.367,148.735
C00729=1103.485,-112.143,-47.182,179.934,4.362,148.733
C00730=1103.490,-112.394,-47.172,179.935,4.357,148.732
C00731=1103.495,-112.643,-47.162,179.936,4.352,148.731
C00732=1103.500,-112.893,-47.153,179.936,4.347,148.729
C00733=1103.506,-113.107,-47.144,179.936,4.342,148.728
C00734=1103.510,-113.322,-47.135,179.936,4.338,148.728
C00735=1103.515,-113.536,-47.127,179.937,4.334,148.726
C00736=1103.518,-113.751,-47.118,179.938,4.330,148.725
C00737=1103.523,-113.965,-47.109,179.938,4.325,148.724
C00738=1103.527,-114.180,-47.101,179.938,4.321,148.723
C00739=1103.532,-114.394,-47.093,179.939,4.316,148.722
C00740=1103.536,-114.609,-47.084,179.939,4.312,148.721
C00741=1103.542,-114.858,-47.074,179.940,4.307,148.720
C00742=1103.548,-115.109,-47.065,179.940,4.302,148.718
C00743=1103.552,-115.358,-47.055,179.941,4.297,148.717
C00744=1103.558,-115.608,-47.044,179.941,4.291,148.716
C00745=1103.563,-115.858,-47.034,179.942,4.287,148.714
C00746=1103.568,-116.107,-47.025,179.943,4.281,148.713
C00747=1103.574,-116.357,-47.015,179.943,4.276,148.712
C00748=1103.578,-116.607,-47.005,179.944,4.271,148.711
C00749=1103.584,-116.857,-46.996,179.944,4.266,148.709
C00750=1103.590,-117.107,-46.985,179.944,4.261,148.708
C00751=1103.595,-117.356,-46.976,179.945,4.256,148.707
C00752=1103.600,-117.606,-46.966,179.946,4.251,148.705
C00753=1103.605,-117.856,-46.956,179.946,4.245,148.704
C00754=1103.610,-118.105,-46.946,179.946,4.240,148.703
C00755=1103.615,-118.355,-46.937,179.947,4.235,148.702
C00756=1103.621,-118.605,-46.927,179.947,4.230,148.700
C00757=1103.627,-118.854,-46.917,179.949,4.225,148.699
C00758=1103.632,-119.104,-46.908,179.949,4.220,148.698
C00759=1103.637,-119.354,-46.897,179.949,4.215,148.696
C00760=1103.642,-119.604,-46.888,179.950,4.209,148.695
C00761=1103.648,-119.854,-46.878,179.950,4.204,148.694
C00762=1103.652,-120.103,-46.869,179.951,4.199,148.693
C00763=1103.658,-120.353,-46.859,179.951,4.193,148.691
C00764=1103.663,-120.602,-46.850,179.952,4.188,148.690
C00765=1103.669,-120.853,-46.840,179.953,4.184,148.689
C00766=1103.673,-121.103,-46.830,179.953,4.178,148.687
C00767=1103.679,-121.353,-46.821,179.954,4.173,148.686
C00768=1103.684,-121.602,-46.811,179.955,4.168,148.684
C00769=1103.690,-121.852,-46.801,179.955,4.162,148.683
C00770=1103.695,-122.101,-46.792,179.955,4.157,148.682
C00771=1103.701,-122.351,-46.782,179.956,4.152,148.681
C00772=1103.706,-122.601,-46.773,179.956,4.147,148.679
C00773=1103.710,-122.851,-46.763,179.957,4.141,148.678
C00774=1103.716,-123.101,-46.753,179.958,4.137,148.677
C00775=1103.721,-123.350,-46.744,179.959,4.131,148.675
C00776=1103.727,-123.600,-46.734,179.959,4.126,148.674
C00777=1103.731,-123.849,-46.725,179.960,4.120,148.673
C00778=1103.737,-124.100,-46.715,179.960,4.115,148.671
C00779=1103.743,-124.350,-46.706,179.961,4.110,148.670
C00780=1103.747,-124.599,-46.697,179.961,4.105,148.669
C00781=1103.753,-124.849,-46.687,179.962,4.099,148.667
C00782=1103.758,-125.098,-46.677,179.962,4.094,148.666
C00783=1103.763,-125.349,-46.668,179.963,4.088,148.664
C00784=1103.768,-125.598,-46.658,179.963,4.083,148.663
C00785=1103.774,-125.848,-46.649,179.964,4.078,148.662
C00786=1103.779,-126.098,-46.640,179.965,4.073,148.661
C00787=1103.784,-126.347,-46.630,179.965,4.067,148.659
C00788=1103.790,-126.598,-46.620,179.966,4.062,148.658
C00789=1103.795,-126.812,-46.612,179.967,4.057,148.657
C00790=1103.798,-127.026,-46.604,179.967,4.053,148.655
C00791=1103.803,-127.241,-46.597,179.968,4.048,148.654
C00792=1103.808,-127.456,-46.588,179.968,4.044,148.653
C00793=1103.812,-127.670,-46.580,179.968,4.039,148.652
C00794=1103.817,-127.885,-46.572,179.969,4.035,148.651
C00795=1103.822,-128.100,-46.564,179.970,4.030,148.649
C00796=1103.826,-128.314,-46.556,179.970,4.025,148.648
C00797=1103.403,-128.304,-46.581,179.978,4.030,148.647
C00798=1103.399,-128.090,-46.590,179.977,4.034,148.648
C00799=1103.394,-127.876,-46.598,179.976,4.039,148.649
C00800=1103.390,-127.661,-46.606,179.976,4.043,148.650
C00801=1103.385,-127.446,-46.614,179.976,4.048,148.652
C00802=1103.380,-127.231,-46.622,179.975,4.053,148.653
C00803=1103.376,-127.017,-46.631,179.974,4.057,148.654
C00804=1103.371,-126.803,-46.639,179.974,4.062,148.655
C00805=1103.366,-126.587,-46.647,179.973,4.066,148.656
C00806=1103.362,-126.338,-46.656,179.973,4.072,148.658
C00807=1103.356,-126.088,-46.665,179.972,4.077,148.659
C00808=1103.351,-125.839,-46.675,179.971,4.082,148.661
C00809=1103.346,-125.589,-46.684,179.971,4.087,148.662
C00810=1103.340,-125.339,-46.694,179.970,4.093,148.663
C00811=1103.335,-125.090,-46.703,179.969,4.099,148.665
C00812=1103.330,-124.840,-46.713,179.969,4.104,148.666
C00813=1103.325,-124.590,-46.723,179.968,4.109,148.667
C00814=1103.320,-124.340,-46.732,179.968,4.114,148.669
C00815=1103.314,-124.090,-46.742,179.967,4.119,148.670
C00816=1103.309,-123.840,-46.751,179.966,4.124,148.671
C00817=1103.303,-123.591,-46.761,179.966,4.129,148.673
C00818=1103.298,-123.341,-46.771,179.965,4.135,148.674
C00819=1103.292,-123.091,-46.780,179.965,4.140,148.675
C00820=1103.288,-122.842,-46.790,179.964,4.146,148.677
C00821=1103.283,-122.592,-46.799,179.964,4.151,148.678
C00822=1103.277,-122.342,-46.809,179.963,4.156,148.679
C00823=1103.272,-122.092,-46.818,179.963,4.161,148.681
C00824=1103.267,-121.843,-46.828,179.962,4.167,148.682
C00825=1103.262,-121.593,-46.837,179.961,4.171,148.683
C00826=1103.256,-121.343,-46.847,179.961,4.177,148.684
C00827=1103.251,-121.093,-46.856,179.960,4.182,148.686
C00828=1103.246,-120.843,-46.867,179.960,4.187,148.687
C00829=1103.241,-120.594,-46.877,179.959,4.193,148.689
C00830=1103.235,-120.344,-46.886,179.959,4.198,148.690
C00831=1103.229,-120.094,-46.896,179.958,4.203,148.691
C00832=1103.224,-119.844,-46.905,179.957,4.208,148.693
C00833=1103.219,-119.595,-46.915,179.957,4.213,148.694
C00834=1103.214,-119.345,-46.925,179.956,4.218,148.695
C00835=1103.208,-119.095,-46.935,179.956,4.224,148.696
C00836=1103.204,-118.845,-46.944,179.955,4.229,148.698
C00837=1103.198,-118.596,-46.955,179.955,4.234,148.699
C00838=1103.193,-118.346,-46.964,179.954,4.239,148.700
C00839=1103.188,-118.096,-46.974,179.953,4.244,148.702
C00840=1103.182,-117.846,-46.984,179.953,4.249,148.703
C00841=1103.177,-117.596,-46.993,179.952,4.254,148.704
C00842=1103.171,-117.347,-47.003,179.952,4.260,148.705
C00843=1103.167,-117.098,-47.013,179.951,4.265,148.707
C00844=1103.161,-116.847,-47.023,179.951,4.270,148.708
C00845=1103.156,-116.597,-47.033,179.950,4.275,148.709
C00846=1103.151,-116.348,-47.043,179.950,4.280,148.711
C00847=1103.145,-116.098,-47.053,179.949,4.285,148.712
C00848=1103.140,-115.849,-47.062,179.949,4.290,148.713
C00849=1103.135,-115.598,-47.072,179.949,4.296,148.714
C00850=1103.129,-115.349,-47.083,179.947,4.300,148.716
C00851=1103.125,-115.100,-47.092,179.947,4.305,148.717
C00852=1103.119,-114.849,-47.102,179.947,4.311,148.718
C00853=1103.114,-114.599,-47.112,179.946,4.316,148.719
C00854=1103.109,-114.385,-47.121,179.946,4.320,148.721
C00855=1103.105,-114.170,-47.129,179.945,4.324,148.722
C00856=1103.100,-113.956,-47.137,179.945,4.329,148.723
C00857=1103.096,-113.742,-47.146,179.945,4.333,148.724
C00858=1103.091,-113.527,-47.155,179.944,4.338,148.725
C00859=1103.087,-113.313,-47.163,179.944,4.342,148.726
C00860=1103.082,-113.098,-47.172,179.943,4.347,148.727
C00861=1103.077,-112.884,-47.180,179.943,4.351,148.728
C00862=1103.073,-112.634,-47.190,179.942,4.356,148.730
C00863=1103.067,-112.384,-47.200,179.942,4.361,148.731
C00864=1103.062,-112.135,-47.211,179.941,4.366,148.732
C00865=1103.056,-111.885,-47.221,179.941,4.371,148.733
C00866=1103.052,-111.635,-47.230,179.941,4.376,148.735
C00867=1103.046,-111.385,-47.240,179.940,4.381,148.736
C00868=1103.040,-111.136,-47.251,179.939,4.386,148.737
C00869=1103.036,-110.886,-47.261,179.939,4.391,148.738
C00870=1103.031,-110.636,-47.271,179.938,4.396,148.740
C00871=1103.025,-110.387,-47.281,179.938,4.401,148.741
C00872=1103.019,-110.137,-47.291,179.937,4.406,148.742
C00873=1103.015,-109.887,-47.301,179.937,4.411,148.743
C00874=1103.010,-109.638,-47.311,179.936,4.416,148.745
C00875=1103.004,-109.387,-47.321,179.936,4.421,148.746
C00876=1102.999,-109.137,-47.331,179.935,4.426,148.747
C00877=1102.994,-108.888,-47.341,179.935,4.431,148.748
C00878=1102.988,-108.638,-47.351,179.934,4.436,148.750
C00879=1102.983,-108.388,-47.362,179.934,4.442,148.751
C00880=1102.978,-108.139,-47.372,179.933,4.446,148.752
C00881=1102.973,-107.889,-47.382,179.933,4.451,148.753
C00882=1102.968,-107.639,-47.392,179.933,4.456,148.755
C00883=1102.962,-107.390,-47.402,179.932,4.461,148.756
C00884=1102.956,-107.140,-47.413,179.932,4.466,148.757
C00885=1102.951,-106.890,-47.423,179.931,4.471,148.758
C00886=1102.947,-106.641,-47.433,179.931,4.476,148.760
C00887=1102.942,-106.390,-47.443,179.930,4.482,148.761
C00888=1102.936,-106.141,-47.454,179.930,4.486,148.762
C00889=1102.930,-105.891,-47.464,179.929,4.491,148.763
C00890=1102.925,-105.641,-47.474,179.929,4.496,148.764
C00891=1102.920,-105.391,-47.485,179.929,4.501,148.766
C00892=1102.915,-105.142,-47.494,179.928,4.506,148.767
C00893=1102.910,-104.892,-47.505,179.928,4.511,148.768
C00894=1102.904,-104.642,-47.515,179.928,4.516,148.769
C00895=1102.899,-104.392,-47.526,179.926,4.521,148.771
C00896=1102.894,-104.143,-47.536,179.926,4.526,148.772
C00897=1102.889,-103.894,-47.547,179.926,4.531,148.773
C00898=1102.884,-103.643,-47.557,179.926,4.536,148.774
C00899=1102.879,-103.394,-47.567,179.925,4.540,148.776
C00900=1102.874,-103.144,-47.577,179.925,4.546,148.777
C00901=1102.868,-102.894,-47.588,179.924,4.551,148.778
C00902=1102.863,-102.644,-47.598,179.923,4.555,148.779
C00903=1102.857,-102.395,-47.608,179.923,4.560,148.780
C00904=1102.852,-102.145,-47.619,179.923,4.565,148.782
C00905=1102.847,-101.895,-47.630,179.923,4.571,148.783
C00906=1102.842,-101.646,-47.640,179.922,4.575,148.784
C00907=1102.837,-101.396,-47.651,179.922,4.580,148.785
C00908=1102.831,-101.146,-47.661,179.922,4.585,148.786
C00909=1102.827,-100.896,-47.671,179.920,4.590,148.788
C00910=1102.822,-100.682,-47.681,179.921,4.595,148.789
C00911=1102.817,-100.468,-47.689,179.920,4.599,148.790
C00912=1102.812,-100.253,-47.699,179.919,4.603,148.791
C00913=1102.808,-100.039,-47.707,179.919,4.607,148.792
C00914=1102.804,-99.824,-47.716,179.919,4.611,148.793
C00915=1102.799,-99.610,-47.725,179.918,4.615,148.794
C00916=1102.795,-99.396,-47.734,179.918,4.620,148.795
C00917=1102.790,-99.181,-47.743,179.918,4.624,148.796
C00918=1102.785,-98.931,-47.754,179.917,4.628,148.797
C00919=1102.780,-98.682,-47.764,179.917,4.633,148.798
C00920=1102.775,-98.432,-47.775,179.917,4.638,148.800
C00921=1102.769,-98.182,-47.785,179.916,4.643,148.801
C00922=1102.765,-97.933,-47.796,179.916,4.648,148.802
C00923=1102.759,-97.683,-47.806,179.916,4.653,148.803
C00924=1102.754,-97.433,-47.817,179.915,4.658,148.804
C00925=1102.748,-97.183,-47.828,179.915,4.663,148.805
C00926=1102.743,-96.933,-47.839,179.914,4.668,148.807
C00927=1102.737,-96.684,-47.849,179.914,4.673,148.808
C00928=1102.732,-96.434,-47.860,179.913,4.677,148.809
C00929=1102.727,-96.185,-47.871,179.913,4.683,148.811
C00930=1102.722,-95.934,-47.881,179.912,4.688,148.812
C00931=1102.717,-95.685,-47.891,179.912,4.692,148.813
C00932=1102.712,-95.435,-47.903,179.911,4.697,148.814
C00933=1102.706,-95.186,-47.913,179.911,4.703,148.815
C00934=1102.701,-94.936,-47.924,179.910,4.707,148.816
C00935=1102.696,-94.687,-47.934,179.910,4.712,148.818
C00936=1102.691,-94.436,-47.945,179.910,4.717,148.819
C00937=1102.685,-94.187,-47.955,179.909,4.721,148.820
C00938=1102.681,-93.937,-47.967,179.909,4.727,148.821
C00939=1102.675,-93.688,-47.977,179.909,4.732,148.822
C00940=1102.670,-93.437,-47.987,179.908,4.736,148.824
C00941=1102.665,-93.188,-47.998,179.908,4.741,148.825
C00942=1102.659,-92.938,-48.009,179.908,4.746,148.826
C00943=1102.654,-92.689,-48.020,179.907,4.752,148.827
C00944=1102.649,-92.439,-48.031,179.907,4.756,148.828
C00945=1102.644,-92.189,-48.042,179.906,4.761,148.830
C00946=1102.639,-91.940,-48.052,179.906,4.766,148.831
C00947=1102.634,-91.689,-48.063,179.906,4.771,148.832
C00948=1102.628,-91.440,-48.074,179.905,4.776,148.833
C00949=1102.623,-91.190,-48.085,179.905,4.781,148.834
C00950=1102.618,-90.941,-48.095,179.905,4.786,148.836
C00951=1102.612,-90.691,-48.107,179.905,4.791,148.837
C00952=1102.608,-90.441,-48.118,179.905,4.796,148.838
C00953=1102.602,-90.192,-48.128,179.904,4.801,148.839
C00954=1102.597,-89.942,-48.139,179.904,4.806,148.840
C00955=1102.592,-89.692,-48.150,179.903,4.811,148.841
C00956=1102.587,-89.443,-48.161,179.903,4.816,148.843
C00957=1102.581,-89.192,-48.172,179.903,4.821,148.844
C00958=1102.576,-88.943,-48.183,179.902,4.825,148.845
C00959=1102.571,-88.693,-48.194,179.902,4.831,148.846
C00960=1102.566,-88.443,-48.205,179.902,4.836,148.847
C00961=1102.561,-88.194,-48.215,179.902,4.841,148.849
C00962=1102.555,-87.944,-48.227,179.901,4.846,148.850
C00963=1102.550,-87.694,-48.237,179.901,4.852,148.851
C00964=1102.545,-87.445,-48.248,179.900,4.856,148.852
C00965=1102.540,-87.195,-48.260,179.900,4.861,148.854
C00966=1102.535,-86.980,-48.269,179.900,4.866,148.855
C00967=1102.531,-86.766,-48.278,179.899,4.870,148.856
C00968=1102.526,-86.552,-48.288,179.899,4.874,148.857
C00969=1102.521,-86.337,-48.297,179.899,4.878,148.858
C00970=1102.517,-86.124,-48.306,179.899,4.883,148.859
C00971=1102.513,-85.909,-48.316,179.898,4.887,148.860
C00972=1102.509,-85.695,-48.325,179.898,4.891,148.861
C00973=1102.504,-85.481,-48.335,179.898,4.896,148.862
C00974=1102.499,-85.231,-48.346,179.898,4.901,148.863
C00975=1102.493,-84.981,-48.358,179.897,4.906,148.864
C00976=1102.489,-84.731,-48.369,179.897,4.911,148.865
C00977=1102.483,-84.481,-48.379,179.897,4.916,148.867
C00978=1102.478,-84.232,-48.390,179.896,4.921,148.868
C00979=1102.473,-83.982,-48.402,179.896,4.926,148.869
C00980=1102.467,-83.732,-48.412,179.896,4.932,148.870
C00981=1102.463,-83.483,-48.424,179.895,4.937,148.872
C00982=1102.457,-83.233,-48.436,179.895,4.942,148.873
C00983=1102.452,-82.984,-48.447,179.895,4.947,148.874
C00984=1102.447,-82.734,-48.457,179.894,4.951,148.875
C00985=1102.442,-82.484,-48.469,179.894,4.957,148.876
C00986=1102.436,-82.235,-48.480,179.894,4.962,148.878
C00987=1102.431,-81.984,-48.490,179.894,4.967,148.879
C00988=1102.426,-81.735,-48.502,179.894,4.972,148.880
C00989=1102.421,-81.485,-48.514,179.894,4.977,148.881
C00990=1102.416,-81.236,-48.525,179.893,4.983,148.882
C00991=1102.410,-80.986,-48.536,179.893,4.988,148.884
C00992=1102.405,-80.736,-48.547,179.893,4.993,148.885
C00993=1102.401,-80.486,-48.558,179.892,4.998,148.886
C00994=1102.395,-80.237,-48.570,179.892,5.003,148.887
C00995=1102.390,-79.987,-48.581,179.892,5.008,148.888
C00996=1102.384,-79.737,-48.592,179.891,5.013,148.890
C00997=1102.380,-79.487,-48.604,179.891,5.018,148.891
C00998=1102.374,-79.238,-48.615,179.891,5.023,148.892
C00999=1102.369,-78.988,-48.626,179.891,5.028,148.893
C01000=1102.364,-78.739,-48.638,179.891,5.033,148.894
C01001=1102.359,-78.489,-48.650,179.890,5.039,148.896
C01002=1102.353,-78.240,-48.661,179.890,5.044,148.897
C01003=1102.348,-77.989,-48.672,179.890,5.049,148.898
C01004=1102.343,-77.740,-48.683,179.890,5.054,148.899
C01005=1102.338,-77.490,-48.695,179.889,5.059,148.900
C01006=1102.332,-77.241,-48.706,179.889,5.064,148.902
C01007=1102.328,-76.991,-48.717,179.889,5.070,148.903
C01008=1102.322,-76.741,-48.729,179.889,5.075,148.904
C01009=1102.317,-76.492,-48.740,179.889,5.080,148.905
C01010=1102.312,-76.242,-48.752,179.889,5.085,148.906
C01011=1102.307,-75.993,-48.763,179.888,5.090,148.907
C01012=1102.301,-75.743,-48.775,179.888,5.095,148.909
C01013=1102.296,-75.493,-48.786,179.888,5.100,148.910
C01014=1102.291,-75.243,-48.797,179.888,5.106,148.911
C01015=1102.286,-74.993,-48.809,179.887,5.110,148.912
C01016=1102.281,-74.743,-48.821,179.887,5.115,148.913
C01017=1102.275,-74.494,-48.831,179.887,5.120,148.915
C01018=1102.270,-74.244,-48.843,179.887,5.125,148.916
C01019=1102.265,-73.994,-48.855,179.887,5.130,148.917
C01020=1102.260,-73.745,-48.867,179.887,5.136,148.918
C01021=1102.254,-73.495,-48.878,179.886,5.141,148.919
C01022=1102.251,-73.281,-48.888,179.887,5.145,148.920
C01023=1102.246,-73.067,-48.898,179.886,5.150,148.921
C01024=1102.241,-72.852,-48.908,179.886,5.154,148.922
C01025=1102.237,-72.638,-48.919,179.886,5.158,148.923
C01026=1102.232,-72.424,-48.928,179.886,5.162,148.924
C01027=1102.228,-72.209,-48.938,179.886,5.167,148.925
C01028=1102.223,-71.996,-48.949,179.886,5.171,148.926
C01029=1102.219,-71.781,-48.959,179.885,5.175,148.927
C01030=1102.214,-71.532,-48.969,179.885,5.181,148.928
C01031=1102.208,-71.282,-48.981,179.885,5.186,148.930
C01032=1102.204,-71.032,-48.993,179.885,5.191,148.931
C01033=1102.198,-70.782,-49.005,179.885,5.196,148.932
C01034=1102.193,-70.533,-49.017,179.885,5.201,148.933
C01035=1102.188,-70.283,-49.028,179.885,5.206,148.934
C01036=1102.183,-70.033,-49.040,179.885,5.211,148.935
C01037=1102.178,-69.784,-49.052,179.885,5.216,148.936
C01038=1102.173,-69.534,-49.063,179.885,5.221,148.937
C01039=1102.167,-69.284,-49.075,179.885,5.226,148.939
C01040=1102.162,-69.035,-49.086,179.884,5.231,148.940
C01041=1102.157,-68.786,-49.099,179.884,5.237,148.941
C01042=1102.152,-68.536,-49.111,179.884,5.242,148.942
C01043=1102.147,-68.286,-49.122,179.885,5.246,148.943
C01044=1102.141,-68.036,-49.134,179.884,5.252,148.944
C01045=1102.136,-67.786,-49.146,179.884,5.257,148.945
C01046=1102.132,-67.537,-49.158,179.884,5.262,148.947
C01047=1102.126,-67.287,-49.170,179.884,5.267,148.948
C01048=1102.121,-67.037,-49.182,179.884,5.272,148.949
C01049=1102.116,-66.788,-49.193,179.884,5.277,148.950
C01050=1102.111,-66.538,-49.206,179.884,5.282,148.951
C01051=1102.106,-66.289,-49.217,179.884,5.287,148.952
C01052=1102.100,-66.039,-49.229,179.884,5.292,148.953
C01053=1102.095,-65.789,-49.241,179.884,5.297,148.954
C01054=1102.090,-65.540,-49.253,179.884,5.302,148.955
C01055=1102.085,-65.290,-49.265,179.884,5.306,148.956
C01056=1102.079,-65.040,-49.277,179.884,5.311,148.958
C01057=1102.075,-64.791,-49.289,179.884,5.316,148.959
C01058=1102.070,-64.541,-49.301,179.884,5.321,148.960
C01059=1102.064,-64.291,-49.313,179.884,5.326,148.961
C01060=1102.059,-64.041,-49.325,179.884,5.331,148.962
C01061=1102.054,-63.792,-49.337,179.884,5.336,148.963
C01062=1102.049,-63.542,-49.349,179.884,5.341,148.964
C01063=1102.044,-63.293,-49.361,179.884,5.346,148.965
C01064=1102.038,-63.043,-49.373,179.884,5.351,148.966
C01065=1102.034,-62.793,-49.384,179.884,5.356,148.967
C01066=1102.029,-62.544,-49.397,179.885,5.361,148.968
C01067=1102.023,-62.294,-49.409,179.885,5.366,148.969
C01068=1102.018,-62.045,-49.421,179.885,5.371,148.970
C01069=1102.013,-61.795,-49.433,179.885,5.376,148.972
C01070=1102.008,-61.545,-49.445,179.885,5.381,148.972
C01071=1102.003,-61.296,-49.457,179.885,5.385,148.974
C01072=1101.997,-61.046,-49.469,179.885,5.390,148.975
C01073=1101.992,-60.796,-49.482,179.885,5.395,148.976
C01074=1101.987,-60.547,-49.494,179.885,5.400,148.977
C01075=1101.982,-60.297,-49.506,179.885,5.405,148.978
C01076=1101.976,-60.047,-49.518,179.885,5.410,148.979
C01077=1101.972,-59.798,-49.530,179.885,5.415,148.980
C01078=1101.967,-59.583,-49.540,179.885,5.419,148.981
C01079=1101.963,-59.369,-49.551,179.885,5.422,148.982
C01080=1101.958,-59.155,-49.562,179.885,5.426,148.982
C01081=1101.954,-58.941,-49.572,179.886,5.431,148.983
C01082=1101.950,-58.726,-49.582,179.885,5.435,148.984
C01083=1101.945,-58.513,-49.593,179.885,5.439,148.985
C01084=1101.941,-58.298,-49.603,179.885,5.443,148.986
C01085=1101.937,-58.084,-49.614,179.885,5.447,148.987
C01086=1101.932,-57.834,-49.626,179.885,5.452,148.988
C01087=1101.926,-57.585,-49.639,179.885,5.456,148.989
C01088=1101.921,-57.335,-49.651,179.884,5.461,148.990
C01089=1101.916,-57.086,-49.663,179.885,5.466,148.991
C01090=1101.911,-56.836,-49.676,179.885,5.471,148.992
C01091=1101.905,-56.586,-49.688,179.884,5.475,148.994
C01092=1101.901,-56.336,-49.701,179.885,5.480,148.994
C01093=1101.895,-56.086,-49.713,179.884,5.485,148.996
C01094=1101.890,-55.837,-49.725,179.884,5.489,148.997
C01095=1101.885,-55.588,-49.738,179.884,5.494,148.998
C01096=1101.880,-55.338,-49.749,179.884,5.499,148.999
C01097=1101.875,-55.089,-49.762,179.884,5.503,149.000
C01098=1101.870,-54.839,-49.773,179.884,5.508,149.001
C01099=1101.865,-54.589,-49.786,179.884,5.513,149.002
C01100=1101.860,-54.340,-49.799,179.883,5.517,149.003
C01101=1101.855,-54.090,-49.811,179.883,5.522,149.004
C01102=1101.850,-53.840,-49.824,179.884,5.527,149.005
C01103=1101.845,-53.591,-49.836,179.883,5.531,149.006
C01104=1101.839,-53.341,-49.848,179.883,5.536,149.007
C01105=1101.835,-53.091,-49.861,179.883,5.541,149.008
C01106=1101.830,-52.842,-49.874,179.883,5.546,149.010
C01107=1101.824,-52.592,-49.887,179.883,5.551,149.011
C01108=1101.818,-52.342,-49.899,179.883,5.555,149.012
C01109=1101.813,-52.093,-49.911,179.883,5.561,149.013
C01110=1101.809,-51.843,-49.924,179.882,5.565,149.014
C01111=1101.803,-51.593,-49.936,179.883,5.570,149.015
C01112=1101.798,-51.344,-49.949,179.883,5.575,149.016
C01113=1101.793,-51.094,-49.961,179.882,5.579,149.017
C01114=1101.788,-50.845,-49.974,179.882,5.584,149.018
C01115=1101.783,-50.595,-49.987,179.882,5.588,149.019
C01116=1101.778,-50.345,-49.999,179.882,5.593,149.020
C01117=1101.773,-50.096,-50.011,179.882,5.598,149.021
C01118=1101.768,-49.846,-50.024,179.881,5.602,149.022
C01119=1101.762,-49.597,-50.037,179.881,5.607,149.024
C01120=1101.758,-49.346,-50.049,179.882,5.612,149.025
C01121=1101.752,-49.097,-50.062,179.881,5.616,149.026
C01122=1101.747,-48.848,-50.075,179.881,5.622,149.027
C01123=1101.742,-48.598,-50.087,179.881,5.626,149.028
C01124=1101.737,-48.348,-50.100,179.881,5.631,149.029
C01125=1101.732,-48.099,-50.113,179.881,5.636,149.030
C01126=1101.727,-47.850,-50.125,179.881,5.640,149.031
C01127=1101.721,-47.600,-50.137,179.880,5.645,149.032
C01128=1101.716,-47.349,-50.151,179.880,5.650,149.033
C01129=1101.711,-47.100,-50.163,179.880,5.655,149.034
C01130=1101.706,-46.851,-50.176,179.880,5.659,149.035
C01131=1101.701,-46.601,-50.189,179.880,5.664,149.037
C01132=1101.696,-46.351,-50.202,179.880,5.669,149.038
C01133=1101.691,-46.102,-50.214,179.880,5.673,149.039
C01134=1101.686,-45.887,-50.226,179.879,5.677,149.040
C01135=1101.682,-45.674,-50.236,179.879,5.681,149.041
C01136=1101.678,-45.460,-50.247,179.879,5.686,149.042
C01137=1101.673,-45.245,-50.258,179.879,5.690,149.042
C01138=1101.669,-45.031,-50.269,179.879,5.694,149.043
C01139=1101.665,-44.817,-50.280,179.879,5.698,149.044
C01140=1101.660,-44.603,-50.291,179.879,5.702,149.045
C01141=1101.656,-44.389,-50.302,179.879,5.706,149.046
C01142=1101.651,-44.140,-50.314,179.879,5.711,149.047
C01143=1101.645,-43.890,-50.328,179.878,5.715,149.048
C01144=1101.640,-43.640,-50.341,179.878,5.720,149.049
C01145=1101.635,-43.391,-50.353,179.878,5.725,149.051
C01146=1101.631,-43.141,-50.366,179.878,5.729,149.052
C01147=1101.625,-42.891,-50.379,179.878,5.734,149.053
C01148=1101.620,-42.642,-50.392,179.878,5.739,149.054
C01149=1101.615,-42.392,-50.405,179.877,5.744,149.055
C01150=1101.610,-42.143,-50.417,179.878,5.748,149.056
C01151=1101.604,-41.893,-50.431,179.878,5.753,149.057
C01152=1101.600,-41.643,-50.444,179.877,5.758,149.058
C01153=1101.594,-41.394,-50.456,179.877,5.762,149.059
C01154=1101.589,-41.144,-50.469,179.877,5.768,149.060
C01155=1101.584,-40.894,-50.482,179.877,5.772,149.061
C01156=1101.579,-40.645,-50.495,179.877,5.777,149.062
C01157=1101.574,-40.395,-50.508,179.878,5.781,149.063
C01158=1101.569,-40.146,-50.522,179.877,5.785,149.064
C01159=1101.564,-39.896,-50.534,179.877,5.790,149.065
C01160=1101.559,-39.646,-50.547,179.877,5.794,149.066
C01161=1101.553,-39.397,-50.561,179.878,5.799,149.067
C01162=1101.548,-39.147,-50.573,179.878,5.804,149.068
C01163=1101.544,-38.897,-50.586,179.878,5.808,149.069
C01164=1101.538,-38.648,-50.599,179.878,5.813,149.070
C01165=1101.533,-38.398,-50.612,179.878,5.818,149.071
C01166=1101.528,-38.149,-50.626,179.878,5.822,149.072
C01167=1101.523,-37.899,-50.639,179.878,5.827,149.073
C01168=1101.518,-37.649,-50.652,179.879,5.831,149.074
C01169=1101.512,-37.400,-50.665,179.878,5.835,149.075
C01170=1101.507,-37.150,-50.678,179.879,5.840,149.076
C01171=1101.503,-36.900,-50.691,179.879,5.844,149.077
C01172=1101.497,-36.651,-50.704,179.879,5.849,149.078
C01173=1101.492,-36.401,-50.717,179.880,5.853,149.078
C01174=1101.487,-36.152,-50.730,179.880,5.857,149.079
C01175=1101.482,-35.902,-50.744,179.880,5.862,149.080
C01176=1101.477,-35.653,-50.757,179.880,5.867,149.081
C01177=1101.471,-35.403,-50.770,179.880,5.871,149.082
C01178=1101.467,-35.153,-50.783,179.881,5.876,149.083
C01179=1101.461,-34.904,-50.796,179.881,5.879,149.084
C01180=1101.457,-34.654,-50.810,179.881,5.884,149.085
C01181=1101.452,-34.405,-50.823,179.881,5.889,149.086
C01182=1101.446,-34.155,-50.836,179.881,5.893,149.087
C01183=1101.442,-33.906,-50.849,179.882,5.898,149.088
C01184=1101.436,-33.656,-50.863,179.882,5.902,149.089
C01185=1101.431,-33.406,-50.876,179.882,5.906,149.089
C01186=1101.426,-33.156,-50.889,179.883,5.911,149.090
C01187=1101.421,-32.907,-50.902,179.883,5.916,149.091
C01188=1101.415,-32.658,-50.916,179.883,5.919,149.092
C01189=1101.411,-32.408,-50.929,179.884,5.924,149.093
C01190=1101.406,-32.194,-50.941,179.884,5.928,149.094
C01191=1101.403,-31.980,-50.952,179.884,5.931,149.094
C01192=1101.398,-31.766,-50.963,179.885,5.936,149.095
C01193=1101.393,-31.552,-50.975,179.885,5.940,149.096
C01194=1101.389,-31.338,-50.986,179.885,5.943,149.097
C01195=1101.384,-31.124,-50.998,179.885,5.947,149.097
C01196=1101.380,-30.910,-51.009,179.885,5.951,149.098
C01197=1101.376,-30.696,-51.021,179.886,5.955,149.099
C01198=1101.371,-30.446,-51.035,179.886,5.959,149.100
C01199=1101.366,-30.197,-51.047,179.887,5.964,149.101
C01200=1101.360,-29.947,-51.061,179.887,5.968,149.102
C01201=1101.356,-29.698,-51.074,179.888,5.973,149.103
C01202=1101.350,-29.448,-51.088,179.887,5.977,149.104
C01203=1101.346,-29.199,-51.101,179.888,5.981,149.104
C01204=1101.340,-28.949,-51.115,179.889,5.986,149.105
C01205=1101.336,-28.699,-51.128,179.889,5.991,149.106
C01206=1101.330,-28.450,-51.142,179.890,5.996,149.107
C01207=1101.325,-28.200,-51.156,179.890,6.000,149.108
C01208=1101.320,-27.951,-51.169,179.890,6.004,149.109
C01209=1101.315,-27.701,-51.183,179.891,6.009,149.110
C01210=1101.310,-27.452,-51.195,179.891,6.014,149.111
C01211=1101.305,-27.202,-51.210,179.891,6.019,149.111
C01212=1101.299,-26.952,-51.223,179.892,6.023,149.112
C01213=1101.295,-26.703,-51.237,179.892,6.028,149.113
C01214=1101.290,-26.452,-51.250,179.893,6.033,149.114
C01215=1101.285,-26.204,-51.263,179.893,6.038,149.115
C01216=1101.280,-25.954,-51.278,179.893,6.043,149.116
C01217=1101.274,-25.704,-51.291,179.894,6.047,149.117
C01218=1101.270,-25.455,-51.305,179.894,6.052,149.118
C01219=1101.265,-25.205,-51.318,179.894,6.056,149.119
C01220=1101.259,-24.956,-51.332,179.894,6.061,149.120
C01221=1101.255,-24.706,-51.346,179.895,6.066,149.121
C01222=1101.250,-24.456,-51.359,179.895,6.070,149.122
C01223=1101.244,-24.207,-51.373,179.895,6.074,149.123
C01224=1101.239,-23.957,-51.388,179.895,6.079,149.124
C01225=1101.234,-23.708,-51.400,179.895,6.084,149.125
C01226=1101.229,-23.458,-51.414,179.896,6.089,149.126
C01227=1101.224,-23.208,-51.428,179.896,6.093,149.127
C01228=1101.219,-22.959,-51.441,179.896,6.098,149.128
C01229=1101.214,-22.709,-51.456,179.896,6.103,149.129
C01230=1101.209,-22.460,-51.470,179.897,6.107,149.130
C01231=1101.203,-22.210,-51.483,179.897,6.111,149.131
C01232=1101.199,-21.961,-51.497,179.897,6.116,149.131
C01233=1101.194,-21.711,-51.511,179.897,6.121,149.133
C01234=1101.188,-21.461,-51.524,179.898,6.126,149.133
C01235=1101.183,-21.212,-51.538,179.897,6.130,149.134
C01236=1101.179,-20.962,-51.552,179.898,6.135,149.135
C01237=1101.173,-20.713,-51.566,179.898,6.139,149.136
C01238=1101.168,-20.463,-51.580,179.899,6.144,149.137
C01239=1101.163,-20.213,-51.594,179.899,6.148,149.138
C01240=1101.158,-19.964,-51.608,179.899,6.153,149.139
C01241=1101.153,-19.715,-51.621,179.900,6.157,149.140
C01242=1101.148,-19.465,-51.636,179.900,6.162,149.141
C01243=1101.143,-19.215,-51.649,179.900,6.166,149.142
C01244=1101.138,-18.966,-51.663,179.900,6.171,149.143
C01245=1101.133,-18.716,-51.678,179.901,6.176,149.144
C01246=1101.126,-18.415,-51.694,179.901,6.181,149.145
C01247=1101.121,-18.112,-51.712,179.902,6.186,149.146
C01248=1101.115,-17.811,-51.728,179.902,6.192,149.147
C01249=1101.108,-17.509,-51.744,179.902,6.197,149.148
C01250=1101.103,-17.259,-51.759,179.903,6.202,149.149
C01251=1101.098,-17.010,-51.773,179.903,6.206,149.150
C01252=1101.093,-16.760,-51.787,179.903,6.211,149.151
C01253=1101.088,-16.511,-51.801,179.904,6.216,149.152
C01254=1101.083,-16.261,-51.815,179.904,6.220,149.152
C01255=1101.078,-16.011,-51.830,179.905,6.225,149.153
C01256=1101.073,-15.761,-51.843,179.905,6.229,149.154
C01257=1101.068,-15.512,-51.857,179.905,6.234,149.155
C01258=1101.063,-15.263,-51.871,179.906,6.238,149.156
C01259=1101.058,-15.013,-51.885,179.906,6.243,149.157
C01260=1101.053,-14.763,-51.899,179.906,6.247,149.158
C01261=1101.048,-14.514,-51.914,179.906,6.252,149.159
C01262=1101.042,-14.265,-51.928,179.907,6.256,149.160
C01263=1101.037,-14.015,-51.942,179.908,6.261,149.160
C01264=1101.033,-13.765,-51.956,179.908,6.265,149.161
C01265=1101.028,-13.515,-51.971,179.908,6.269,149.162
C01266=1101.023,-13.266,-51.985,179.909,6.274,149.163
C01267=1101.017,-13.017,-51.999,179.909,6.279,149.164
C01268=1101.012,-12.767,-52.013,179.910,6.284,149.165
C01269=1101.007,-12.517,-52.027,179.910,6.287,149.166
C01270=1101.002,-12.268,-52.042,179.910,6.292,149.167
C01271=1100.998,-12.019,-52.057,179.911,6.297,149.167
C01272=1100.992,-11.770,-52.070,179.912,6.301,149.168
C01273=1100.987,-11.520,-52.085,179.912,6.306,149.169
C01274=1100.982,-11.270,-52.099,179.912,6.310,149.170
C01275=1100.977,-11.020,-52.113,179.913,6.315,149.171
C01276=1100.972,-10.771,-52.128,179.913,6.319,149.172
C01277=1100.967,-10.521,-52.142,179.914,6.324,149.172
C01278=1100.962,-10.271,-52.156,179.915,6.328,149.173
C01279=1100.957,-10.022,-52.170,179.914,6.332,149.174
C01280=1100.952,-9.773,-52.185,179.915,6.337,149.175
C01281=1100.947,-9.523,-52.199,179.915,6.342,149.176
C01282=1100.942,-9.274,-52.214,179.916,6.346,149.177
C01283=1100.937,-9.024,-52.228,179.917,6.351,149.178
C01284=1100.932,-8.774,-52.242,179.917,6.355,149.179
C01285=1100.927,-8.525,-52.256,179.917,6.359,149.179
C01286=1100.923,-8.276,-52.271,179.918,6.364,149.180
C01287=1100.917,-8.027,-52.285,179.919,6.368,149.181
C01288=1100.912,-7.777,-52.300,179.919,6.373,149.182
C01289=1100.907,-7.527,-52.314,179.920,6.378,149.183
C01290=1100.901,-7.277,-52.329,179.920,6.383,149.184
C01291=1100.897,-7.028,-52.344,179.921,6.386,149.184
C01292=1100.892,-6.778,-52.358,179.921,6.391,149.185
C01293=1100.887,-6.529,-52.372,179.922,6.396,149.186
C01294=1100.882,-6.279,-52.387,179.922,6.400,149.187
C01295=1100.877,-6.030,-52.402,179.923,6.405,149.188
C01296=1100.872,-5.780,-52.416,179.924,6.409,149.189
C01297=1100.867,-5.530,-52.431,179.924,6.414,149.190
C01298=1100.640,-15.232,-51.913,179.911,6.242,149.155
C01299=1100.646,-15.481,-51.899,179.911,6.237,149.154
C01300=1100.651,-15.731,-51.885,179.911,6.233,149.153
C01301=1100.656,-15.981,-51.871,179.910,6.228,149.152
C01302=1100.661,-16.230,-51.856,179.910,6.224,149.152
C01303=1100.666,-16.479,-51.842,179.909,6.219,149.151
C01304=1100.671,-16.729,-51.828,179.909,6.215,149.150
C01305=1100.676,-16.979,-51.814,179.908,6.211,149.149
C01306=1100.681,-17.229,-51.801,179.908,6.206,149.148
C01307=1100.689,-17.598,-51.780,179.907,6.199,149.147
C01308=1100.696,-17.969,-51.759,179.907,6.192,149.145
C01309=1100.704,-18.339,-51.738,179.906,6.185,149.144
C01310=1100.711,-18.709,-51.717,179.906,6.179,149.143
C01311=1100.716,-18.958,-51.703,179.906,6.174,149.142
C01312=1100.721,-19.208,-51.690,179.905,6.170,149.141
C01313=1100.726,-19.458,-51.676,179.906,6.165,149.140
C01314=1100.731,-19.707,-51.661,179.905,6.161,149.139
C01315=1100.736,-19.957,-51.647,179.905,6.156,149.138
C01316=1100.741,-20.206,-51.634,179.904,6.151,149.137
C01317=1100.746,-20.456,-51.619,179.904,6.147,149.136
C01318=1100.751,-20.706,-51.606,179.904,6.143,149.135
C01319=1100.757,-20.955,-51.592,179.903,6.138,149.134
C01320=1100.762,-21.205,-51.578,179.903,6.133,149.133
C01321=1100.766,-21.454,-51.564,179.903,6.129,149.133
C01322=1100.772,-21.704,-51.551,179.903,6.124,149.131
C01323=1100.777,-21.953,-51.537,179.903,6.119,149.131
C01324=1100.782,-22.203,-51.522,179.902,6.115,149.130
C01325=1100.787,-22.452,-51.509,179.902,6.111,149.129
C01326=1100.792,-22.702,-51.495,179.902,6.106,149.128
C01327=1100.797,-22.952,-51.481,179.902,6.101,149.127
C01328=1100.802,-23.201,-51.467,179.901,6.096,149.126
C01329=1100.807,-23.451,-51.454,179.901,6.092,149.125
C01330=1100.812,-23.701,-51.440,179.901,6.087,149.124
C01331=1100.817,-23.950,-51.426,179.901,6.083,149.123
C01332=1100.823,-24.200,-51.412,179.901,6.078,149.122
C01333=1100.828,-24.449,-51.399,179.901,6.074,149.121
C01334=1100.832,-24.698,-51.385,179.900,6.069,149.120
C01335=1100.838,-24.949,-51.371,179.900,6.064,149.119
C01336=1100.843,-25.197,-51.358,179.900,6.060,149.118
C01337=1100.848,-25.447,-51.344,179.900,6.055,149.117
C01338=1100.853,-25.697,-51.330,179.899,6.051,149.116
C01339=1100.858,-25.946,-51.317,179.899,6.045,149.115
C01340=1100.863,-26.196,-51.303,179.899,6.041,149.114
C01341=1100.868,-26.445,-51.289,179.898,6.036,149.113
C01342=1100.873,-26.695,-51.276,179.898,6.031,149.112
C01343=1100.878,-26.945,-51.262,179.897,6.026,149.111
C01344=1100.883,-27.194,-51.248,179.897,6.022,149.111
C01345=1100.888,-27.444,-51.235,179.897,6.017,149.110
C01346=1100.894,-27.693,-51.221,179.896,6.012,149.109
C01347=1100.898,-27.943,-51.207,179.896,6.008,149.108
C01348=1100.904,-28.192,-51.194,179.896,6.004,149.107
C01349=1100.909,-28.442,-51.180,179.895,5.999,149.106
C01350=1100.913,-28.692,-51.167,179.895,5.994,149.105
C01351=1100.919,-28.941,-51.153,179.894,5.989,149.104
C01352=1100.923,-29.191,-51.140,179.894,5.985,149.103
C01353=1100.929,-29.440,-51.126,179.893,5.980,149.103
C01354=1100.934,-29.690,-51.113,179.893,5.976,149.102
C01355=1100.939,-29.940,-51.100,179.893,5.972,149.101
C01356=1100.944,-30.189,-51.086,179.892,5.967,149.100
C01357=1100.949,-30.439,-51.073,179.892,5.962,149.099
C01358=1100.954,-30.688,-51.059,179.891,5.958,149.098
C01359=1100.958,-30.903,-51.048,179.891,5.954,149.097
C01360=1100.963,-31.116,-51.036,179.891,5.950,149.096
C01361=1100.967,-31.330,-51.024,179.891,5.947,149.096
C01362=1100.971,-31.545,-51.014,179.890,5.943,149.095
C01363=1100.976,-31.759,-51.002,179.890,5.938,149.094
C01364=1100.980,-31.971,-50.991,179.890,5.935,149.094
C01365=1100.985,-32.186,-50.979,179.889,5.931,149.093
C01366=1100.989,-32.400,-50.967,179.889,5.927,149.092
C01367=1100.994,-32.650,-50.954,179.889,5.923,149.091
C01368=1101.000,-32.900,-50.941,179.889,5.919,149.090
C01369=1101.004,-33.149,-50.927,179.888,5.914,149.089
C01370=1101.010,-33.399,-50.914,179.888,5.910,149.088
C01371=1101.014,-33.649,-50.901,179.888,5.906,149.088
C01372=1101.020,-33.898,-50.887,179.887,5.901,149.087
C01373=1101.024,-34.148,-50.874,179.887,5.896,149.086
C01374=1101.030,-34.397,-50.861,179.887,5.892,149.085
C01375=1101.034,-34.647,-50.847,179.887,5.887,149.084
C01376=1101.039,-34.896,-50.835,179.886,5.883,149.083
C01377=1101.045,-35.146,-50.822,179.886,5.879,149.082
C01378=1101.049,-35.395,-50.808,179.886,5.874,149.081
C01379=1101.055,-35.645,-50.795,179.885,5.869,149.080
C01380=1101.060,-35.895,-50.782,179.886,5.865,149.079
C01381=1101.066,-36.144,-50.769,179.885,5.861,149.078
C01382=1101.070,-36.394,-50.755,179.885,5.857,149.078
C01383=1101.075,-36.643,-50.742,179.885,5.852,149.077
C01384=1101.080,-36.893,-50.729,179.884,5.847,149.076
C01385=1101.085,-37.143,-50.716,179.884,5.843,149.075
C01386=1101.091,-37.392,-50.702,179.884,5.839,149.074
C01387=1101.096,-37.642,-50.689,179.884,5.835,149.073
C01388=1101.101,-37.891,-50.677,179.884,5.830,149.072
C01389=1101.106,-38.141,-50.663,179.884,5.825,149.071
C01390=1101.111,-38.391,-50.650,179.884,5.821,149.070
C01391=1101.117,-38.640,-50.637,179.883,5.816,149.069
C01392=1101.121,-38.890,-50.624,179.883,5.811,149.068
C01393=1101.126,-39.139,-50.611,179.884,5.807,149.067
C01394=1101.132,-39.389,-50.597,179.883,5.802,149.066
C01395=1101.137,-39.639,-50.585,179.883,5.798,149.065
C01396=1101.142,-39.888,-50.572,179.883,5.793,149.064
C01397=1101.147,-40.138,-50.559,179.883,5.789,149.063
C01398=1101.152,-40.388,-50.546,179.883,5.785,149.062
C01399=1101.157,-40.636,-50.533,179.883,5.780,149.061
C01400=1101.162,-40.887,-50.519,179.883,5.776,149.060
C01401=1101.167,-41.136,-50.507,179.883,5.771,149.059
C01402=1101.172,-41.386,-50.494,179.883,5.766,149.058
C01403=1101.178,-41.636,-50.480,179.884,5.761,149.057
C01404=1101.183,-41.885,-50.468,179.883,5.757,149.056
C01405=1101.187,-42.135,-50.455,179.883,5.752,149.055
C01406=1101.193,-42.384,-50.442,179.884,5.747,149.054
C01407=1101.198,-42.634,-50.429,179.883,5.743,149.053
C01408=1101.203,-42.884,-50.416,179.884,5.737,149.052
C01409=1101.208,-43.133,-50.403,179.884,5.733,149.051
C01410=1101.213,-43.383,-50.391,179.884,5.728,149.049
C01411=1101.218,-43.633,-50.377,179.884,5.724,149.048
C01412=1101.224,-43.882,-50.365,179.884,5.719,149.047
C01413=1101.229,-44.132,-50.352,179.885,5.714,149.046
C01414=1101.233,-44.382,-50.339,179.885,5.710,149.045
C01415=1101.239,-44.595,-50.328,179.885,5.706,149.044
C01416=1101.242,-44.809,-50.317,179.885,5.701,149.043
C01417=1101.246,-45.023,-50.306,179.885,5.697,149.042
C01418=1101.251,-45.238,-50.295,179.885,5.693,149.041
C01419=1101.256,-45.451,-50.284,179.885,5.689,149.040
C01420=1101.260,-45.666,-50.273,179.886,5.685,149.039
C01421=1101.264,-45.880,-50.262,179.886,5.681,149.039
C01422=1101.268,-46.094,-50.251,179.886,5.677,149.038
C01423=1101.273,-46.343,-50.238,179.886,5.672,149.036
C01424=1101.279,-46.593,-50.225,179.886,5.667,149.036
C01425=1101.284,-46.843,-50.212,179.886,5.663,149.034
C01426=1101.289,-47.093,-50.200,179.886,5.658,149.033
C01427=1101.294,-47.342,-50.188,179.887,5.654,149.032
C01428=1101.299,-47.591,-50.175,179.887,5.649,149.031
C01429=1101.304,-47.841,-50.162,179.887,5.644,149.030
C01430=1101.310,-48.091,-50.149,179.887,5.639,149.029
C01431=1101.315,-48.340,-50.136,179.887,5.635,149.028
C01432=1101.320,-48.590,-50.124,179.887,5.630,149.027
C01433=1101.325,-48.840,-50.111,179.888,5.625,149.026
C01434=1101.330,-49.089,-50.098,179.888,5.620,149.025
C01435=1101.335,-49.339,-50.086,179.887,5.615,149.024
C01436=1101.340,-49.588,-50.074,179.888,5.611,149.022
C01437=1101.345,-49.838,-50.060,179.888,5.606,149.021
C01438=1101.351,-50.088,-50.047,179.888,5.601,149.020
C01439=1101.356,-50.337,-50.035,179.888,5.597,149.019
C01440=1101.361,-50.587,-50.023,179.888,5.592,149.018
C01441=1101.366,-50.837,-50.010,179.888,5.587,149.017
C01442=1101.371,-51.086,-49.997,179.889,5.583,149.016
C01443=1101.376,-51.336,-49.985,179.889,5.578,149.015
C01444=1101.381,-51.585,-49.972,179.888,5.573,149.014
C01445=1101.386,-51.835,-49.960,179.889,5.569,149.013
C01446=1101.391,-52.085,-49.947,179.889,5.563,149.012
C01447=1101.396,-52.334,-49.935,179.889,5.559,149.011
C01448=1101.402,-52.584,-49.922,179.889,5.554,149.010
C01449=1101.407,-52.834,-49.910,179.889,5.549,149.008
C01450=1101.413,-53.083,-49.897,179.889,5.545,149.007
C01451=1101.417,-53.333,-49.884,179.890,5.540,149.006
C01452=1101.423,-53.583,-49.872,179.889,5.535,149.005
C01453=1101.428,-53.832,-49.860,179.889,5.530,149.004
C01454=1101.433,-54.082,-49.847,179.890,5.526,149.003
C01455=1101.438,-54.331,-49.834,179.890,5.521,149.002
C01456=1101.443,-54.581,-49.823,179.890,5.516,149.001
C01457=1101.448,-54.831,-49.810,179.890,5.512,149.000
C01458=1101.453,-55.080,-49.797,179.890,5.507,148.999
C01459=1101.458,-55.330,-49.785,179.890,5.502,148.998
C01460=1101.464,-55.580,-49.773,179.890,5.498,148.997
C01461=1101.469,-55.829,-49.760,179.890,5.493,148.996
C01462=1101.474,-56.079,-49.748,179.890,5.488,148.994
C01463=1101.479,-56.329,-49.735,179.891,5.484,148.994
C01464=1101.484,-56.579,-49.723,179.891,5.479,148.992
C01465=1101.488,-56.828,-49.711,179.891,5.474,148.991
C01466=1101.494,-57.077,-49.699,179.890,5.469,148.990
C01467=1101.499,-57.327,-49.687,179.891,5.465,148.989
C01468=1101.504,-57.576,-49.674,179.891,5.460,148.988
C01469=1101.510,-57.826,-49.662,179.891,5.455,148.987
C01470=1101.514,-58.076,-49.649,179.891,5.451,148.986
C01471=1101.519,-58.290,-49.639,179.891,5.447,148.985
C01472=1101.523,-58.504,-49.628,179.891,5.442,148.984
C01473=1101.528,-58.719,-49.618,179.891,5.438,148.983
C01474=1101.532,-58.933,-49.607,179.891,5.434,148.982
C01475=1101.536,-59.147,-49.596,179.891,5.430,148.981
C01476=1101.541,-59.361,-49.586,179.892,5.426,148.981
C01477=1101.545,-59.575,-49.575,179.892,5.422,148.980
C01478=1101.549,-59.790,-49.565,179.891,5.418,148.979
C01479=1101.555,-60.039,-49.553,179.892,5.414,148.978
C01480=1101.560,-60.289,-49.541,179.892,5.409,148.977
C01481=1101.565,-60.538,-49.528,179.891,5.404,148.976
C01482=1101.571,-60.788,-49.516,179.891,5.399,148.975
C01483=1101.575,-61.037,-49.504,179.891,5.394,148.974
C01484=1101.580,-61.287,-49.493,179.891,5.389,148.972
C01485=1101.585,-61.536,-49.480,179.891,5.384,148.971
C01486=1101.591,-61.786,-49.468,179.891,5.379,148.970
C01487=1101.596,-62.036,-49.455,179.890,5.374,148.969
C01488=1101.601,-62.286,-49.444,179.891,5.369,148.968
C01489=1101.606,-62.535,-49.432,179.890,5.364,148.967
C01490=1101.611,-62.785,-49.420,179.891,5.360,148.966
C01491=1101.617,-63.035,-49.408,179.891,5.355,148.965
C01492=1101.621,-63.285,-49.395,179.891,5.350,148.964
C01493=1101.627,-63.534,-49.383,179.891,5.345,148.963
C01494=1101.631,-63.784,-49.372,179.890,5.340,148.962
C01495=1101.636,-64.033,-49.359,179.890,5.335,148.961
C01496=1101.642,-64.283,-49.347,179.891,5.330,148.960
C01497=1101.647,-64.533,-49.335,179.890,5.325,148.959
C01498=1101.652,-64.782,-49.323,179.890,5.320,148.958
C01499=1101.657,-65.032,-49.311,179.890,5.315,148.956
C01500=1101.662,-65.282,-49.299,179.890,5.310,148.955
C01501=1101.668,-65.532,-49.287,179.890,5.305,148.954
C01502=1101.673,-65.781,-49.275,179.890,5.300,148.953
C01503=1101.678,-66.030,-49.263,179.890,5.295,148.952
C01504=1101.683,-66.280,-49.251,179.890,5.290,148.951
C01505=1101.688,-66.530,-49.239,179.891,5.286,148.950
C01506=1101.693,-66.780,-49.228,179.891,5.281,148.949
C01507=1101.698,-67.029,-49.215,179.891,5.276,148.948
C01508=1101.704,-67.279,-49.203,179.891,5.271,148.947
C01509=1101.709,-67.529,-49.192,179.891,5.266,148.945
C01510=1101.714,-67.778,-49.181,179.891,5.260,148.944
C01511=1101.719,-68.027,-49.168,179.891,5.255,148.943
C01512=1101.725,-68.277,-49.156,179.891,5.251,148.942
C01513=1101.730,-68.527,-49.145,179.891,5.245,148.941
C01514=1101.735,-68.777,-49.133,179.891,5.240,148.940
C01515=1101.740,-69.027,-49.121,179.891,5.235,148.939
C01516=1101.745,-69.276,-49.109,179.891,5.230,148.937
C01517=1101.750,-69.526,-49.097,179.891,5.225,148.936
C01518=1101.756,-69.776,-49.085,179.891,5.220,148.935
C01519=1101.760,-70.025,-49.074,179.891,5.215,148.934
C01520=1101.766,-70.275,-49.062,179.891,5.210,148.933
C01521=1101.771,-70.525,-49.050,179.891,5.205,148.932
C01522=1101.776,-70.774,-49.038,179.891,5.200,148.931
C01523=1101.781,-71.024,-49.026,179.892,5.195,148.929
C01524=1101.786,-71.273,-49.015,179.892,5.189,148.928
C01525=1101.792,-71.523,-49.004,179.892,5.184,148.927
C01526=1101.797,-71.773,-48.992,179.892,5.179,148.926
C01527=1101.801,-71.987,-48.981,179.892,5.175,148.925
C01528=1101.805,-72.201,-48.972,179.892,5.171,148.924
C01529=1101.810,-72.416,-48.962,179.892,5.166,148.923
C01530=1101.814,-72.629,-48.952,179.893,5.162,148.922
C01531=1101.819,-72.844,-48.942,179.893,5.158,148.921
C01532=1101.824,-73.058,-48.932,179.893,5.153,148.920
C01533=1101.828,-73.273,-48.921,179.893,5.150,148.919
C01534=1101.833,-73.487,-48.912,179.893,5.144,148.918
C01535=1101.837,-73.736,-48.900,179.893,5.139,148.917
C01536=1101.843,-73.986,-48.888,179.893,5.134,148.916
C01537=1101.847,-74.236,-48.877,179.893,5.129,148.914
C01538=1101.853,-74.485,-48.866,179.894,5.124,148.913
C01539=1101.858,-74.735,-48.854,179.894,5.120,148.912
C01540=1101.864,-74.985,-48.842,179.894,5.114,148.911
C01541=1101.868,-75.234,-48.831,179.895,5.109,148.910
C01542=1101.874,-75.484,-48.819,179.895,5.104,148.909
C01543=1101.879,-75.734,-48.807,179.895,5.099,148.907
C01544=1101.884,-75.983,-48.796,179.895,5.094,148.906
C01545=1101.890,-76.233,-48.785,179.895,5.089,148.905
C01546=1101.895,-76.483,-48.773,179.895,5.084,148.904
C01547=1101.900,-76.733,-48.761,179.896,5.078,148.903
C01548=1101.905,-76.982,-48.750,179.896,5.073,148.902
C01549=1101.911,-77.232,-48.739,179.896,5.068,148.900
C01550=1101.915,-77.481,-48.727,179.896,5.063,148.899
C01551=1101.920,-77.731,-48.716,179.896,5.058,148.898
C01552=1101.926,-77.981,-48.705,179.896,5.053,148.897
C01553=1101.931,-78.231,-48.694,179.896,5.048,148.896
C01554=1101.937,-78.480,-48.682,179.897,5.042,148.894
C01555=1101.941,-78.730,-48.671,179.897,5.037,148.893
C01556=1101.947,-78.980,-48.659,179.897,5.032,148.892
C01557=1101.951,-79.229,-48.648,179.898,5.027,148.891
C01558=1101.957,-79.479,-48.636,179.898,5.022,148.890
C01559=1101.962,-79.728,-48.625,179.899,5.017,148.888
C01560=1101.968,-79.979,-48.614,179.899,5.012,148.887
C01561=1101.973,-80.228,-48.602,179.899,5.007,148.886
C01562=1101.977,-80.478,-48.591,179.899,5.002,148.885
C01563=1101.983,-80.727,-48.579,179.899,4.997,148.884
C01564=1101.988,-80.977,-48.568,179.899,4.992,148.882
C01565=1101.993,-81.227,-48.558,179.899,4.986,148.881
C01566=1101.998,-81.477,-48.546,179.900,4.981,148.880
C01567=1102.004,-81.726,-48.535,179.900,4.976,148.879
C01568=1102.009,-81.976,-48.523,179.900,4.971,148.878
C01569=1102.014,-82.226,-48.512,179.901,4.965,148.876
C01570=1102.019,-82.475,-48.501,179.901,4.961,148.875
C01571=1102.025,-82.725,-48.490,179.902,4.956,148.874
C01572=1102.030,-82.975,-48.478,179.902,4.951,148.873
C01573=1102.034,-83.224,-48.467,179.902,4.946,148.872
C01574=1102.041,-83.474,-48.456,179.902,4.941,148.870
C01575=1102.045,-83.724,-48.445,179.902,4.935,148.869
C01576=1102.050,-83.973,-48.434,179.903,4.930,148.868
C01577=1102.056,-84.223,-48.423,179.903,4.925,148.867
C01578=1102.061,-84.473,-48.411,179.903,4.920,148.865
C01579=1102.066,-84.723,-48.400,179.903,4.915,148.864
C01580=1102.072,-84.972,-48.389,179.904,4.910,148.863
C01581=1102.077,-85.222,-48.378,179.904,4.905,148.862
C01582=1102.081,-85.472,-48.367,179.905,4.900,148.861
C01583=1102.086,-85.686,-48.357,179.905,4.895,148.860
C01584=1102.090,-85.900,-48.348,179.905,4.891,148.859
C01585=1102.095,-86.115,-48.338,179.905,4.887,148.858
C01586=1102.100,-86.329,-48.328,179.906,4.883,148.856
C01587=1102.103,-86.543,-48.319,179.906,4.878,148.855
C01588=1102.108,-86.757,-48.309,179.906,4.874,148.855
C01589=1102.113,-86.972,-48.301,179.907,4.870,148.853
C01590=1102.117,-87.187,-48.291,179.906,4.865,148.852
C01591=1102.122,-87.436,-48.280,179.907,4.860,148.851
C01592=1102.127,-87.685,-48.269,179.907,4.855,148.850
C01593=1102.133,-87.936,-48.258,179.908,4.850,148.849
C01594=1102.138,-88.185,-48.247,179.908,4.845,148.848
C01595=1102.143,-88.435,-48.236,179.908,4.839,148.846
C01596=1102.148,-88.684,-48.225,179.909,4.834,148.845
C01597=1102.153,-88.934,-48.215,179.909,4.829,148.844
C01598=1102.159,-89.184,-48.203,179.910,4.825,148.843
C01599=1102.164,-89.433,-48.192,179.910,4.820,148.841
C01600=1102.169,-89.683,-48.181,179.910,4.815,148.840
C01601=1102.174,-89.933,-48.170,179.910,4.809,148.839
C01602=1102.179,-90.182,-48.160,179.910,4.804,148.838
C01603=1102.185,-90.432,-48.148,179.911,4.800,148.837
C01604=1102.190,-90.682,-48.138,179.911,4.795,148.836
C01605=1102.195,-90.932,-48.126,179.912,4.790,148.834
C01606=1102.200,-91.182,-48.116,179.912,4.785,148.833
C01607=1102.205,-91.431,-48.105,179.912,4.779,148.832
C01608=1102.210,-91.681,-48.094,179.913,4.775,148.831
C01609=1102.216,-91.930,-48.083,179.913,4.770,148.830
C01610=1102.221,-92.180,-48.072,179.913,4.765,148.828
C01611=1102.226,-92.431,-48.062,179.913,4.760,148.827
C01612=1102.232,-92.680,-48.051,179.914,4.755,148.826
C01613=1102.237,-92.930,-48.040,179.914,4.750,148.825
C01614=1102.242,-93.179,-48.029,179.914,4.745,148.824
C01615=1102.247,-93.429,-48.019,179.915,4.740,148.822
C01616=1102.252,-93.678,-48.008,179.915,4.736,148.821
C01617=1102.257,-93.928,-47.997,179.916,4.730,148.820
C01618=1102.263,-94.179,-47.986,179.916,4.725,148.819
C01619=1102.268,-94.428,-47.975,179.917,4.721,148.818
C01620=1102.273,-94.678,-47.965,179.917,4.716,148.816
C01621=1102.279,-94.927,-47.954,179.917,4.711,148.815
C01622=1102.284,-95.177,-47.943,179.918,4.706,148.814
C01623=1102.289,-95.427,-47.933,179.918,4.701,148.813
C01624=1102.294,-95.676,-47.922,179.918,4.696,148.812
C01625=1102.300,-95.926,-47.911,179.919,4.692,148.810
C01626=1102.305,-96.176,-47.901,179.919,4.687,148.809
C01627=1102.310,-96.425,-47.890,179.919,4.681,148.808
C01628=1102.315,-96.675,-47.879,179.920,4.677,148.807
C01629=1102.320,-96.925,-47.869,179.920,4.672,148.806
C01630=1102.325,-97.174,-47.858,179.921,4.667,148.805
C01631=1102.331,-97.424,-47.848,179.921,4.662,148.803
C01632=1102.336,-97.674,-47.837,179.922,4.657,148.802
C01633=1102.341,-97.924,-47.827,179.922,4.652,148.801
C01634=1102.346,-98.173,-47.815,179.923,4.647,148.799
C01635=1102.352,-98.423,-47.805,179.923,4.642,148.798
C01636=1102.357,-98.673,-47.795,179.924,4.637,148.797
C01637=1102.362,-98.922,-47.784,179.924,4.632,148.796
C01638=1102.367,-99.172,-47.773,179.925,4.628,148.795
C01639=1102.372,-99.387,-47.764,179.925,4.624,148.794
C01640=1102.376,-99.601,-47.755,179.925,4.619,148.793
C01641=1102.381,-99.815,-47.746,179.925,4.615,148.792
C01642=1102.385,-100.030,-47.737,179.926,4.611,148.791
C01643=1102.389,-100.244,-47.728,179.926,4.607,148.790
C01644=1102.395,-100.459,-47.719,179.927,4.602,148.788
C01645=1102.399,-100.673,-47.710,179.927,4.598,148.788
C01646=1102.404,-100.887,-47.701,179.927,4.594,148.787
C01647=1102.409,-101.138,-47.690,179.928,4.589,148.785
C01648=1102.414,-101.386,-47.680,179.928,4.584,148.784
C01649=1102.419,-101.637,-47.669,179.929,4.579,148.783
C01650=1102.424,-101.886,-47.659,179.929,4.574,148.782
C01651=1102.429,-102.136,-47.649,179.930,4.569,148.780
C01652=1102.435,-102.386,-47.638,179.930,4.564,148.779
C01653=1102.440,-102.636,-47.628,179.930,4.559,148.778
C01654=1102.445,-102.885,-47.617,179.931,4.555,148.777
C01655=1102.451,-103.135,-47.607,179.931,4.549,148.776
C01656=1102.456,-103.385,-47.596,179.931,4.544,148.774
C01657=1102.461,-103.634,-47.586,179.932,4.540,148.773
C01658=1102.466,-103.885,-47.575,179.932,4.535,148.772
C01659=1102.471,-104.134,-47.566,179.933,4.530,148.771
C01660=1102.477,-104.383,-47.556,179.933,4.524,148.769
C01661=1102.482,-104.634,-47.545,179.934,4.520,148.768
C01662=1102.487,-104.883,-47.534,179.934,4.515,148.767
C01663=1102.492,-105.133,-47.523,179.935,4.509,148.766
C01664=1102.498,-105.382,-47.513,179.936,4.505,148.764
C01665=1102.503,-105.632,-47.503,179.936,4.500,148.763
C01666=1102.508,-105.882,-47.493,179.936,4.495,148.762
C01667=1102.513,-106.131,-47.483,179.936,4.490,148.761
C01668=1102.518,-106.382,-47.472,179.937,4.485,148.760
C01669=1102.524,-106.631,-47.462,179.937,4.480,148.758
C01670=1102.529,-106.881,-47.452,179.938,4.475,148.757
C01671=1102.534,-107.131,-47.441,179.939,4.470,148.756
C01672=1102.539,-107.380,-47.432,179.939,4.465,148.755
C01673=1102.544,-107.630,-47.421,179.939,4.460,148.753
C01674=1102.550,-107.880,-47.411,179.940,4.455,148.752
C01675=1102.555,-108.130,-47.401,179.940,4.451,148.751
C01676=1102.560,-108.380,-47.390,179.941,4.445,148.750
C01677=1102.565,-108.629,-47.381,179.941,4.440,148.749
C01678=1102.571,-108.879,-47.370,179.942,4.435,148.747
C01679=1102.576,-109.129,-47.360,179.942,4.430,148.746
C01680=1102.581,-109.378,-47.350,179.943,4.425,148.745
C01681=1102.587,-109.628,-47.339,179.943,4.420,148.743
C01682=1102.591,-109.878,-47.329,179.943,4.415,148.742
C01683=1102.597,-110.127,-47.319,179.944,4.411,148.741
C01684=1102.602,-110.377,-47.309,179.945,4.405,148.740
C01685=1102.607,-110.627,-47.298,179.945,4.400,148.738
C01686=1102.613,-110.877,-47.289,179.945,4.395,148.737
C01687=1102.618,-111.127,-47.279,179.946,4.390,148.736
C01688=1102.623,-111.377,-47.269,179.946,4.385,148.735
C01689=1102.629,-111.626,-47.258,179.947,4.380,148.733
C01690=1102.634,-111.876,-47.249,179.947,4.375,148.732
C01691=1102.639,-112.125,-47.239,179.948,4.369,148.731
C01692=1102.644,-112.375,-47.228,179.949,4.365,148.730
C01693=1102.649,-112.625,-47.218,179.949,4.360,148.728
C01694=1102.655,-112.875,-47.209,179.950,4.354,148.727
C01695=1102.659,-113.089,-47.200,179.950,4.350,148.726
C01696=1102.664,-113.303,-47.192,179.951,4.346,148.725
C01697=1102.668,-113.519,-47.182,179.950,4.341,148.724
C01698=1102.673,-113.733,-47.174,179.951,4.337,148.723
C01699=1102.677,-113.947,-47.166,179.952,4.333,148.722
C01700=1102.682,-114.161,-47.157,179.952,4.329,148.720
C01701=1102.686,-114.376,-47.148,179.952,4.324,148.719
C01702=1102.691,-114.590,-47.140,179.953,4.320,148.718
C01703=1102.696,-114.840,-47.130,179.953,4.314,148.717
C01704=1102.702,-115.089,-47.120,179.954,4.310,148.716
C01705=1102.706,-115.340,-47.110,179.955,4.305,148.714
C01706=1102.712,-115.589,-47.100,179.955,4.299,148.713
C01707=1102.718,-115.839,-47.090,179.955,4.294,148.712
C01708=1102.722,-116.088,-47.080,179.956,4.289,148.711
C01709=1102.728,-116.339,-47.070,179.957,4.284,148.709
C01710=1102.733,-116.589,-47.060,179.957,4.279,148.708
C01711=1102.738,-116.838,-47.051,179.958,4.274,148.707
C01712=1102.744,-117.087,-47.040,179.958,4.269,148.705
C01713=1102.748,-117.338,-47.031,179.959,4.263,148.704
C01714=1102.754,-117.587,-47.021,179.959,4.258,148.703
C01715=1102.760,-117.837,-47.011,179.960,4.254,148.702
C01716=1102.765,-118.087,-47.002,179.961,4.248,148.700
C01717=1102.770,-118.336,-46.992,179.961,4.243,148.699
C01718=1102.775,-118.586,-46.982,179.962,4.238,148.698
C01719=1102.780,-118.837,-46.972,179.962,4.233,148.696
C01720=1102.786,-119.086,-46.962,179.962,4.227,148.695
C01721=1102.791,-119.335,-46.952,179.964,4.223,148.694
C01722=1102.797,-119.585,-46.943,179.964,4.218,148.693
C01723=1102.801,-119.835,-46.933,179.964,4.212,148.691
C01724=1102.807,-120.085,-46.923,179.965,4.207,148.690
C01725=1102.812,-120.335,-46.914,179.965,4.202,148.689
C01726=1102.817,-120.584,-46.903,179.966,4.196,148.687
C01727=1102.822,-120.834,-46.894,179.966,4.191,148.686
C01728=1102.828,-121.084,-46.884,179.967,4.187,148.685
C01729=1102.833,-121.334,-46.874,179.968,4.181,148.683
C01730=1102.838,-121.584,-46.865,179.968,4.176,148.682
C01731=1102.844,-121.833,-46.855,179.969,4.170,148.681
C01732=1102.849,-122.083,-46.845,179.969,4.165,148.679
C01733=1102.855,-122.333,-46.836,179.970,4.160,148.678
C01734=1102.860,-122.582,-46.826,179.971,4.155,148.677
C01735=1102.865,-122.833,-46.816,179.971,4.149,148.675
C01736=1102.870,-123.082,-46.806,179.972,4.145,148.674
C01737=1102.875,-123.332,-46.798,179.972,4.140,148.673
C01738=1102.881,-123.581,-46.787,179.973,4.134,148.671
C01739=1102.885,-123.831,-46.778,179.974,4.129,148.670
C01740=1102.891,-124.081,-46.768,179.974,4.123,148.669
C01741=1102.896,-124.330,-46.759,179.975,4.118,148.667
C01742=1102.902,-124.580,-46.749,179.975,4.113,148.666
C01743=1102.906,-124.830,-46.739,179.976,4.108,148.665
C01744=1102.912,-125.080,-46.730,179.977,4.102,148.663
C01745=1102.917,-125.330,-46.720,179.977,4.097,148.662
C01746=1102.923,-125.580,-46.711,179.978,4.091,148.661
C01747=1102.928,-125.829,-46.701,179.979,4.087,148.659
C01748=1102.933,-126.079,-46.692,179.979,4.081,148.658
C01749=1102.939,-126.329,-46.683,179.980,4.076,148.656
C01750=1102.944,-126.578,-46.673,179.981,4.071,148.655
C01751=1102.948,-126.793,-46.665,179.981,4.066,148.654
C01752=1102.953,-127.007,-46.656,179.982,4.061,148.653
C01753=1102.958,-127.222,-46.649,179.982,4.057,148.652
C01754=1102.962,-127.437,-46.640,179.982,4.052,148.650
C01755=1102.967,-127.651,-46.632,179.983,4.048,148.649
C01756=1102.971,-127.866,-46.624,179.984,4.043,148.648
C01757=1102.976,-128.081,-46.616,179.984,4.038,148.647
C01758=1102.980,-128.295,-46.608,179.985,4.034,148.646
C01759=1102.558,-128.285,-46.633,179.992,4.038,148.644
C01760=1102.553,-128.071,-46.642,179.992,4.043,148.646
C01761=1102.548,-127.856,-46.650,179.991,4.047,148.647
C01762=1102.544,-127.642,-46.658,179.991,4.052,148.648
C01763=1102.539,-127.427,-46.666,179.990,4.056,148.649
C01764=1102.535,-127.212,-46.674,179.989,4.061,148.650
C01765=1102.530,-126.998,-46.683,179.989,4.066,148.651
C01766=1102.526,-126.783,-46.691,179.988,4.070,148.653
C01767=1102.521,-126.570,-46.699,179.988,4.074,148.654
C01768=1102.516,-126.319,-46.708,179.987,4.080,148.655
C01769=1102.510,-126.070,-46.718,179.986,4.085,148.657
C01770=1102.505,-125.820,-46.727,179.986,4.090,148.658
C01771=1102.500,-125.570,-46.738,179.985,4.096,148.659
C01772=1102.494,-125.320,-46.746,179.985,4.101,148.661
C01773=1102.489,-125.071,-46.757,179.984,4.107,148.662
C01774=1102.484,-124.821,-46.766,179.983,4.112,148.663
C01775=1102.479,-124.572,-46.775,179.983,4.117,148.665
C01776=1102.474,-124.321,-46.785,179.982,4.123,148.666
C01777=1102.469,-124.072,-46.795,179.982,4.128,148.667
C01778=1102.463,-123.821,-46.804,179.981,4.132,148.669
C01779=1102.458,-123.572,-46.814,179.980,4.138,148.670
C01780=1102.452,-123.323,-46.824,179.980,4.143,148.671
C01781=1102.447,-123.073,-46.833,179.979,4.149,148.673
C01782=1102.442,-122.823,-46.843,179.978,4.154,148.674
C01783=1102.437,-122.573,-46.852,179.978,4.159,148.675
C01784=1102.431,-122.323,-46.862,179.977,4.164,148.677
C01785=1102.427,-122.074,-46.872,179.977,4.170,148.678
C01786=1102.421,-121.824,-46.882,179.976,4.174,148.679
C01787=1102.415,-121.574,-46.892,179.975,4.179,148.681
C01788=1102.410,-121.324,-46.901,179.975,4.185,148.682
C01789=1102.405,-121.074,-46.911,179.974,4.190,148.683
C01790=1102.400,-120.825,-46.921,179.974,4.196,148.685
C01791=1102.394,-120.575,-46.930,179.973,4.201,148.686
C01792=1102.389,-120.326,-46.940,179.972,4.206,148.687
C01793=1102.384,-120.076,-46.950,179.972,4.211,148.689
C01794=1102.379,-119.825,-46.959,179.971,4.216,148.690
C01795=1102.373,-119.576,-46.970,179.971,4.221,148.691
C01796=1102.368,-119.326,-46.980,179.970,4.227,148.693
C01797=1102.363,-119.077,-46.989,179.970,4.232,148.694
C01798=1102.357,-118.827,-46.999,179.969,4.237,148.695
C01799=1102.353,-118.577,-47.009,179.968,4.242,148.696
C01800=1102.347,-118.327,-47.019,179.968,4.247,148.698
C01801=1102.341,-118.077,-47.029,179.967,4.252,148.699
C01802=1102.336,-117.828,-47.038,179.967,4.257,148.700
C01803=1102.331,-117.578,-47.049,179.966,4.263,148.702
C01804=1102.326,-117.328,-47.058,179.966,4.268,148.703
C01805=1102.321,-117.078,-47.068,179.965,4.272,148.704
C01806=1102.315,-116.829,-47.078,179.964,4.278,148.706
C01807=1102.310,-116.580,-47.088,179.964,4.283,148.707
C01808=1102.305,-116.329,-47.098,179.964,4.288,148.708
C01809=1102.299,-116.079,-47.108,179.963,4.293,148.709
C01810=1102.294,-115.830,-47.117,179.962,4.298,148.711
C01811=1102.289,-115.581,-47.128,179.962,4.303,148.712
C01812=1102.284,-115.330,-47.138,179.962,4.308,148.713
C01813=1102.279,-115.080,-47.147,179.961,4.314,148.715
C01814=1102.273,-114.831,-47.157,179.961,4.319,148.716
C01815=1102.268,-114.581,-47.168,179.960,4.323,148.717
C01816=1102.264,-114.366,-47.176,179.959,4.329,148.718
C01817=1102.259,-114.152,-47.185,179.959,4.333,148.719
C01818=1102.255,-113.938,-47.194,179.958,4.337,148.720
C01819=1102.250,-113.723,-47.202,179.958,4.341,148.721
C01820=1102.246,-113.509,-47.210,179.958,4.346,148.723
C01821=1102.241,-113.294,-47.219,179.957,4.350,148.724
C01822=1102.236,-113.080,-47.228,179.957,4.354,148.725
C01823=1102.232,-112.866,-47.237,179.956,4.358,148.726
C01824=1102.226,-112.616,-47.247,179.956,4.363,148.727
C01825=1102.222,-112.366,-47.257,179.955,4.369,148.728
C01826=1102.216,-112.116,-47.266,179.955,4.374,148.730
C01827=1102.211,-111.867,-47.276,179.954,4.378,148.731
C01828=1102.206,-111.616,-47.287,179.954,4.384,148.732
C01829=1102.201,-111.367,-47.297,179.953,4.389,148.734
C01830=1102.195,-111.118,-47.307,179.953,4.394,148.735
C01831=1102.190,-110.867,-47.317,179.952,4.399,148.736
C01832=1102.185,-110.618,-47.328,179.952,4.404,148.737
C01833=1102.180,-110.369,-47.337,179.951,4.409,148.738
C01834=1102.175,-110.118,-47.348,179.951,4.414,148.740
C01835=1102.169,-109.869,-47.358,179.950,4.419,148.741
C01836=1102.163,-109.619,-47.368,179.950,4.424,148.742
C01837=1102.158,-109.369,-47.379,179.949,4.429,148.743
C01838=1102.154,-109.120,-47.388,179.949,4.434,148.745
C01839=1102.148,-108.870,-47.399,179.948,4.439,148.746
